LIN {X 0,Y 207.652,Z 346.509,A -85,B 0,C 180,E1 -25427.031,E2 -25427.031} C_VEL
LIN {X 0,Y 210.503,Z 352.306,A -85,B 0,C 180,E1 -25428.836,E2 -25428.836} C_VEL
LIN {X 0,Y 203.288,Z 423.819,A -85,B 0,C 180,E1 -25430.749,E2 -25430.749} C_VEL
LIN {X 0,Y 200.381,Z 440.802,A -85,B 0,C 180,E1 -25431.417,E2 -25431.417} C_VEL
LIN {X 0,Y 196.445,Z 457.536,A -85,B 0,C 180,E1 -25432.38,E2 -25432.38} C_VEL
LIN {X 0,Y 191.604,Z 473.562,A -85,B 0,C 180,E1 -25433.622,E2 -25433.622} C_VEL
LIN {X 0,Y 186.062,Z 488.689,A -85,B 0,C 180,E1 -25435.158,E2 -25435.158} C_VEL
LIN {X 0,Y 179.509,Z 503.688,A -85,B 0,C 180,E1 -25437.096,E2 -25437.096} C_VEL
LIN {X 0,Y 172.547,Z 517.473,A -85,B 0,C 180,E1 -25439.393,E2 -25439.393} C_VEL
LIN {X 0,Y 164.589,Z 531.208,A -85,B 0,C 180,E1 -25442.33,E2 -25442.33} C_VEL
LIN {X 0,Y 157.144,Z 542.82,A -85,B 0,C 180,E1 -25445.563,E2 -25445.563} C_VEL
LIN {X 0,Y 149.721,Z 553.398,A -85,B 0,C 180,E1 -25449.305,E2 -25449.305} C_VEL
LIN {X 0,Y 142.748,Z 562.767,A -85,B 0,C 180,E1 -25453.554,E2 -25453.554} C_VEL
LIN {X 0,Y 136.314,Z 570.972,A -85,B 0,C 180,E1 -25458.403,E2 -25458.403} C_VEL
LIN {X 0,Y 130.699,Z 578.07,A -85,B 0,C 180,E1 -25463.825,E2 -25463.825} C_VEL
LIN {X 0,Y 125.94,Z 584.277,A -85,B 0,C 180,E1 -25469.999,E2 -25469.999} C_VEL
LIN {X 0,Y 122.402,Z 589.195,A -85,B 0,C 180,E1 -25476.593,E2 -25476.593} C_VEL
LIN {X 0,Y 119.976,Z 592.988,A -85,B 0,C 180,E1 -25483.55,E2 -25483.55} C_VEL
LIN {X 0,Y 118.782,Z 595.717,A -85,B 0,C 180,E1 -25490.792,E2 -25490.792} C_VEL
LIN {X 0,Y 118.646,Z 597.115,A -85,B 0,C 180,E1 -25497.312,E2 -25497.312} C_VEL
LIN {X 0,Y 119.339,Z 597.749,A -85,B 0,C 180,E1 -25504.465,E2 -25504.465} C_VEL
LIN {X 0,Y 120.964,Z 597.343,A -85,B 0,C 180,E1 -25510.949,E2 -25510.949} C_VEL
LIN {X 0,Y 123.876,Z 596.092,A -85,B 0,C 180,E1 -25517.521,E2 -25517.521} C_VEL
LIN {X 0,Y 128.898,Z 593.311,A -85,B 0,C 180,E1 -25524.868,E2 -25524.868} C_VEL
LIN {X 0,Y 135.659,Z 589.135,A -85,B 0,C 180,E1 -25531.725,E2 -25531.725} C_VEL
LIN {X 0,Y 144.193,Z 583.478,A -85,B 0,C 180,E1 -25537.826,E2 -25537.826} C_VEL
LIN {X 0,Y 152.82,Z 577.234,A -85,B 0,C 180,E1 -25542.598,E2 -25542.598} C_VEL
LIN {X 0,Y 163.268,Z 568.849,A -85,B 0,C 180,E1 -25547.195,E2 -25547.195} C_VEL
LIN {X 0,Y 174.835,Z 558.387,A -85,B 0,C 180,E1 -25551.263,E2 -25551.263} C_VEL
LIN {X 0,Y 185.382,Z 547.58,A -85,B 0,C 180,E1 -25554.346,E2 -25554.346} C_VEL
LIN {X 0,Y 195.153,Z 536.256,A -85,B 0,C 180,E1 -25556.791,E2 -25556.791} C_VEL
LIN {X 0,Y 204.724,Z 523.645,A -85,B 0,C 180,E1 -25558.892,E2 -25558.892} C_VEL
LIN {X 0,Y 213.483,Z 510.379,A -85,B 0,C 180,E1 -25560.609,E2 -25560.609} C_VEL
LIN {X 0,Y 220.417,Z 498.375,A -85,B 0,C 180,E1 -25561.827,E2 -25561.827} C_VEL
LIN {X 0,Y 227.397,Z 484.222,A -85,B 0,C 180,E1 -25562.988,E2 -25562.988} C_VEL
LIN {X 0,Y 233.808,Z 468.556,A -85,B 0,C 180,E1 -25564.007,E2 -25564.007} C_VEL
LIN {X 0,Y 239.121,Z 452.344,A -85,B 0,C 180,E1 -25564.783,E2 -25564.783} C_VEL
LIN {X 0,Y 243.235,Z 435.804,A -85,B 0,C 180,E1 -25565.349,E2 -25565.349} C_VEL
LIN {X 0,Y 246.105,Z 418.602,A -85,B 0,C 180,E1 -25565.773,E2 -25565.773} C_VEL
LIN {X 0,Y 251.259,Z 376.905,A -85,B 0,C 180,E1 -25566.684,E2 -25566.684} C_VEL
LIN {X 0,Y 250.782,Z 375.19,A -85,B 0,C 180,E1 -25568.055,E2 -25568.055} C_VEL
LIN {X 0,Y 250.079,Z 372.447,A -85,B 0,C 180,E1 -25572.163,E2 -25572.163} C_VEL
LIN {X 0,Y 250.037,Z 372.701,A -85,B 0,C 180,E1 -25573.31,E2 -25573.31} C_VEL
LIN {X 0,Y 250.756,Z 375.692,A -85,B 0,C 180,E1 -25577.654,E2 -25577.654} C_VEL
LIN {X 0,Y 251.253,Z 377.3,A -85,B 0,C 180,E1 -25579.03,E2 -25579.03} C_VEL
LIN {X 0,Y 244.616,Z 429.393,A -85,B 0,C 180,E1 -25580.146,E2 -25580.146} C_VEL
LIN {X 0,Y 241.029,Z 446.475,A -85,B 0,C 180,E1 -25580.592,E2 -25580.592} C_VEL
LIN {X 0,Y 236.395,Z 462.41,A -85,B 0,C 180,E1 -25581.149,E2 -25581.149} C_VEL
LIN {X 0,Y 230.959,Z 477.274,A -85,B 0,C 180,E1 -25581.862,E2 -25581.862} C_VEL
LIN {X 0,Y 224.757,Z 491.347,A -85,B 0,C 180,E1 -25582.717,E2 -25582.717} C_VEL
LIN {X 0,Y 217.928,Z 504.427,A -85,B 0,C 180,E1 -25583.787,E2 -25583.787} C_VEL
LIN {X 0,Y 208.905,Z 519.27,A -85,B 0,C 180,E1 -25585.296,E2 -25585.296} C_VEL
LIN {X 0,Y 200.844,Z 530.92,A -85,B 0,C 180,E1 -25586.838,E2 -25586.838} C_VEL
LIN {X 0,Y 190.88,Z 543.575,A -85,B 0,C 180,E1 -25589.023,E2 -25589.023} C_VEL
LIN {X 0,Y 181.232,Z 554.346,A -85,B 0,C 180,E1 -25591.448,E2 -25591.448} C_VEL
LIN {X 0,Y 170.694,Z 564.923,A -85,B 0,C 180,E1 -25594.57,E2 -25594.57} C_VEL
LIN {X 0,Y 169.098,Z 566.423,A -85,B 0,C 180,E1 -25595.081,E2 -25595.081} C_VEL
LIN {X 0,Y 165.201,Z 569.732,A -85,B 0,C 180,E1 -25596.102,E2 -25596.102} C_VEL
LIN {X 0,Y 157.698,Z 574.973,A -85,B 0,C 180,E1 -25597.464,E2 -25597.464} C_VEL
LIN {X 0,Y 150.146,Z 579.765,A -85,B 0,C 180,E1 -25599.042,E2 -25599.042} C_VEL
LIN {X 0,Y 146.248,Z 582.367,A -85,B 0,C 180,E1 -25600.426,E2 -25600.426} C_VEL
LIN {X 0,Y 136.237,Z 589.443,A -85,B 0,C 180,E1 -25605.862,E2 -25605.862} C_VEL
LIN {X 0,Y 128.84,Z 594.26,A -85,B 0,C 180,E1 -25611.15,E2 -25611.15} C_VEL
LIN {X 0,Y 121.309,Z 598.92,A -85,B 0,C 180,E1 -25618.575,E2 -25618.575} C_VEL
LIN {X 0,Y 116.893,Z 601.559,A -85,B 0,C 180,E1 -25625.112,E2 -25625.112} C_VEL
LIN {X 0,Y 113.834,Z 603.26,A -85,B 0,C 180,E1 -25632.021,E2 -25632.021} C_VEL
LIN {X 0,Y 112.343,Z 604.035,A -85,B 0,C 180,E1 -25639.184,E2 -25639.184} C_VEL
LIN {X 0,Y 112.095,Z 603.898,A -85,B 0,C 180,E1 -25646.406,E2 -25646.406} C_VEL
LIN {X 0,Y 112.259,Z 603.468,A -85,B 0,C 180,E1 -25650.001,E2 -25650.001} C_VEL
LIN {X 0,Y 112.154,Z 602.73,A -85,B 0,C 180,E1 -25653.594,E2 -25653.594} C_VEL
LIN {X 0,Y 112.377,Z 600.537,A -85,B 0,C 180,E1 -25660.815,E2 -25660.815} C_VEL
LIN {X 0,Y 113.815,Z 597.25,A -85,B 0,C 180,E1 -25667.985,E2 -25667.985} C_VEL
LIN {X 0,Y 116.648,Z 592.834,A -85,B 0,C 180,E1 -25674.946,E2 -25674.946} C_VEL
LIN {X 0,Y 120.876,Z 587.27,A -85,B 0,C 180,E1 -25681.553,E2 -25681.553} C_VEL
LIN {X 0,Y 126.437,Z 580.31,A -85,B 0,C 180,E1 -25687.694,E2 -25687.694} C_VEL
LIN {X 0,Y 133.293,Z 571.931,A -85,B 0,C 180,E1 -25693.27,E2 -25693.27} C_VEL
LIN {X 0,Y 141.317,Z 561.914,A -85,B 0,C 180,E1 -25698.244,E2 -25698.244} C_VEL
LIN {X 0,Y 148.682,Z 551.934,A -85,B 0,C 180,E1 -25702.085,E2 -25702.085} C_VEL
LIN {X 0,Y 157.311,Z 539.305,A -85,B 0,C 180,E1 -25705.741,E2 -25705.741} C_VEL
LIN {X 0,Y 165.607,Z 525.855,A -85,B 0,C 180,E1 -25708.656,E2 -25708.656} C_VEL
LIN {X 0,Y 172.473,Z 513.183,A -85,B 0,C 180,E1 -25710.8,E2 -25710.8} C_VEL
LIN {X 0,Y 179.768,Z 497.842,A -85,B 0,C 180,E1 -25712.799,E2 -25712.799} C_VEL
LIN {X 0,Y 185.354,Z 483.986,A -85,B 0,C 180,E1 -25714.226,E2 -25714.226} C_VEL
LIN {X 0,Y 190.733,Z 468.038,A -85,B 0,C 180,E1 -25715.46,E2 -25715.46} C_VEL
LIN {X 0,Y 194.945,Z 452.39,A -85,B 0,C 180,E1 -25716.337,E2 -25716.337} C_VEL
LIN {X 0,Y 198.282,Z 436,A -85,B 0,C 180,E1 -25716.992,E2 -25716.992} C_VEL
LIN {X 0,Y 200.576,Z 417.694,A -85,B 0,C 180,E1 -25717.565,E2 -25717.565} C_VEL
LIN {X 0,Y 206.676,Z 357.209,A -85,B 0,C 180,E1 -25719.155,E2 -25719.155} C_VEL
LIN {X 0,Y 203.434,Z 349.128,A -85,B 0,C 180,E1 -25721.494,E2 -25721.494} C_VEL
LIN {X 0,Y 198.655,Z 340.024,A -85,B 0,C 180,E1 -25725.138,E2 -25725.138} C_VEL
LIN {X 0,Y 195.269,Z 333.943,A -85,B 0,C 180,E1 -25728.08,E2 -25728.08} C_VEL
LIN {X 0,Y 192.367,Z 328.903,A -85,B 0,C 180,E1 -25730.999,E2 -25730.999} C_VEL
LIN {X 0,Y 189.117,Z 323.394,A -85,B 0,C 180,E1 -25734.828,E2 -25734.828} C_VEL
LIN {X 0,Y 186.858,Z 319.626,A -85,B 0,C 180,E1 -25738.137,E2 -25738.137} C_VEL
LIN {X 0,Y 184.729,Z 315.82,A -85,B 0,C 180,E1 -25742.307,E2 -25742.307} C_VEL
LIN {X 0,Y 184.223,Z 315.108,A -85,B 0,C 180,E1 -25743.467,E2 -25743.467} C_VEL
LIN {X 0,Y 182.713,Z 313.172,A -85,B 0,C 180,E1 -25748.571,E2 -25748.571} C_VEL
LIN {X 0,Y 182.415,Z 311.657,A -85,B 0,C 180,E1 -25752.151,E2 -25752.151} C_VEL
LIN {X 0,Y 182.382,Z 311.95,A -85,B 0,C 180,E1 -25754.436,E2 -25754.436} C_VEL
LIN {X 0,Y 183.988,Z 315.501,A -85,B 0,C 180,E1 -25762.686,E2 -25762.686} C_VEL
LIN {X 0,Y 184.724,Z 316.384,A -85,B 0,C 180,E1 -25764.365,E2 -25764.365} C_VEL
LIN {X 0,Y 187.441,Z 320.995,A -85,B 0,C 180,E1 -25769.378,E2 -25769.378} C_VEL
LIN {X 0,Y 190.002,Z 325.194,A -85,B 0,C 180,E1 -25772.883,E2 -25772.883} C_VEL
LIN {X 0,Y 193.097,Z 330.301,A -85,B 0,C 180,E1 -25776.321,E2 -25776.321} C_VEL
LIN {X 0,Y 197.341,Z 337.624,A -85,B 0,C 180,E1 -25780.284,E2 -25780.284} C_VEL
LIN {X 0,Y 202.688,Z 347.63,A -85,B 0,C 180,E1 -25784.496,E2 -25784.496} C_VEL
LIN {X 0,Y 206.664,Z 355.706,A -85,B 0,C 180,E1 -25787.241,E2 -25787.241} C_VEL
LIN {X 0,Y 199.416,Z 424.921,A -85,B 0,C 180,E1 -25789.058,E2 -25789.058} C_VEL
LIN {X 0,Y 196.238,Z 442.746,A -85,B 0,C 180,E1 -25789.777,E2 -25789.777} C_VEL
LIN {X 0,Y 192.185,Z 459.017,A -85,B 0,C 180,E1 -25790.721,E2 -25790.721} C_VEL
LIN {X 0,Y 187.194,Z 474.829,A -85,B 0,C 180,E1 -25791.956,E2 -25791.956} C_VEL
LIN {X 0,Y 181.535,Z 489.677,A -85,B 0,C 180,E1 -25793.471,E2 -25793.471} C_VEL
LIN {X 0,Y 174.797,Z 504.536,A -85,B 0,C 180,E1 -25795.395,E2 -25795.395} C_VEL
LIN {X 0,Y 167.766,Z 518.005,A -85,B 0,C 180,E1 -25797.639,E2 -25797.639} C_VEL
LIN {X 0,Y 160.036,Z 530.9,A -85,B 0,C 180,E1 -25800.393,E2 -25800.393} C_VEL
LIN {X 0,Y 152.843,Z 541.768,A -85,B 0,C 180,E1 -25803.363,E2 -25803.363} C_VEL
LIN {X 0,Y 144.749,Z 552.984,A -85,B 0,C 180,E1 -25807.295,E2 -25807.295} C_VEL
LIN {X 0,Y 136.71,Z 563.26,A -85,B 0,C 180,E1 -25812.034,E2 -25812.034} C_VEL
LIN {X 0,Y 129.48,Z 572.063,A -85,B 0,C 180,E1 -25817.46,E2 -25817.46} C_VEL
LIN {X 0,Y 123.401,Z 579.326,A -85,B 0,C 180,E1 -25823.459,E2 -25823.459} C_VEL
LIN {X 0,Y 118.554,Z 585.3,A -85,B 0,C 180,E1 -25829.999,E2 -25829.999} C_VEL
LIN {X 0,Y 114.968,Z 590.109,A -85,B 0,C 180,E1 -25837.021,E2 -25837.021} C_VEL
LIN {X 0,Y 112.606,Z 593.693,A -85,B 0,C 180,E1 -25844.456,E2 -25844.456} C_VEL
LIN {X 0,Y 111.836,Z 595.471,A -85,B 0,C 180,E1 -25849.502,E2 -25849.502} C_VEL
LIN {X 0,Y 111.555,Z 597.357,A -85,B 0,C 180,E1 -25858.115,E2 -25858.115} C_VEL
LIN {X 0,Y 112.415,Z 597.959,A -85,B 0,C 180,E1 -25865.636,E2 -25865.636} C_VEL
LIN {X 0,Y 114.335,Z 597.539,A -85,B 0,C 180,E1 -25872.542,E2 -25872.542} C_VEL
LIN {X 0,Y 118.302,Z 595.932,A -85,B 0,C 180,E1 -25880.558,E2 -25880.558} C_VEL
LIN {X 0,Y 124.144,Z 593.005,A -85,B 0,C 180,E1 -25888.119,E2 -25888.119} C_VEL
LIN {X 0,Y 131.806,Z 588.593,A -85,B 0,C 180,E1 -25895.016,E2 -25895.016} C_VEL
LIN {X 0,Y 141.166,Z 582.701,A -85,B 0,C 180,E1 -25901.066,E2 -25901.066} C_VEL
LIN {X 0,Y 151.88,Z 575.162,A -85,B 0,C 180,E1 -25906.34,E2 -25906.34} C_VEL
LIN {X 0,Y 162.15,Z 567.093,A -85,B 0,C 180,E1 -25910.309,E2 -25910.309} C_VEL
LIN {X 0,Y 173.171,Z 557.354,A -85,B 0,C 180,E1 -25913.873,E2 -25913.873} C_VEL
LIN {X 0,Y 183.061,Z 547.566,A -85,B 0,C 180,E1 -25916.523,E2 -25916.523} C_VEL
LIN {X 0,Y 193.3,Z 535.996,A -85,B 0,C 180,E1 -25918.912,E2 -25918.912} C_VEL
LIN {X 0,Y 203.056,Z 523.461,A -85,B 0,C 180,E1 -25920.91,E2 -25920.91} C_VEL
LIN {X 0,Y 211.921,Z 510.362,A -85,B 0,C 180,E1 -25922.536,E2 -25922.536} C_VEL
LIN {X 0,Y 219.769,Z 496.993,A -85,B 0,C 180,E1 -25923.801,E2 -25923.801} C_VEL
LIN {X 0,Y 227.299,Z 481.61,A -85,B 0,C 180,E1 -25924.97,E2 -25924.97} C_VEL
LIN {X 0,Y 233.568,Z 466.034,A -85,B 0,C 180,E1 -25925.864,E2 -25925.864} C_VEL
LIN {X 0,Y 238.605,Z 450.348,A -85,B 0,C 180,E1 -25926.553,E2 -25926.553} C_VEL
LIN {X 0,Y 242.42,Z 434.847,A -85,B 0,C 180,E1 -25927.037,E2 -25927.037} C_VEL
LIN {X 0,Y 245.308,Z 417.581,A -85,B 0,C 180,E1 -25927.434,E2 -25927.434} C_VEL
LIN {X 0,Y 249.773,Z 382.182,A -85,B 0,C 180,E1 -25928.18,E2 -25928.18} C_VEL
LIN {X 0,Y 249.115,Z 379.534,A -85,B 0,C 180,E1 -25932.211,E2 -25932.211} C_VEL
LIN {X 0,Y 249.072,Z 380.047,A -85,B 0,C 180,E1 -25933.68,E2 -25933.68} C_VEL
LIN {X 0,Y 249.662,Z 382.544,A -85,B 0,C 180,E1 -25937.298,E2 -25937.298} C_VEL
LIN {X 0,Y 249.721,Z 382.826,A -85,B 0,C 180,E1 -25937.517,E2 -25937.517} C_VEL
LIN {X 0,Y 243.632,Z 429.235,A -85,B 0,C 180,E1 -25938.491,E2 -25938.491} C_VEL
LIN {X 0,Y 239.964,Z 446.328,A -85,B 0,C 180,E1 -25938.916,E2 -25938.916} C_VEL
LIN {X 0,Y 235.154,Z 462.482,A -85,B 0,C 180,E1 -25939.445,E2 -25939.445} C_VEL
LIN {X 0,Y 229.275,Z 478.077,A -85,B 0,C 180,E1 -25940.16,E2 -25940.16} C_VEL
LIN {X 0,Y 222.96,Z 491.964,A -85,B 0,C 180,E1 -25940.965,E2 -25940.965} C_VEL
LIN {X 0,Y 215.992,Z 504.967,A -85,B 0,C 180,E1 -25941.98,E2 -25941.98} C_VEL
LIN {X 0,Y 207.556,Z 518.518,A -85,B 0,C 180,E1 -25943.3,E2 -25943.3} C_VEL
LIN {X 0,Y 197.782,Z 532.101,A -85,B 0,C 180,E1 -25945.029,E2 -25945.029} C_VEL
LIN {X 0,Y 187.573,Z 544.548,A -85,B 0,C 180,E1 -25947.146,E2 -25947.146} C_VEL
LIN {X 0,Y 177.657,Z 555.179,A -85,B 0,C 180,E1 -25949.509,E2 -25949.509} C_VEL
LIN {X 0,Y 166.777,Z 565.552,A -85,B 0,C 180,E1 -25952.565,E2 -25952.565} C_VEL
LIN {X 0,Y 156.514,Z 574.365,A -85,B 0,C 180,E1 -25956.076,E2 -25956.076} C_VEL
LIN {X 0,Y 146.248,Z 582.367,A -85,B 0,C 180,E1 -25960.426,E2 -25960.426} C_VEL
LIN {X 0,Y 142.37,Z 584.882,A -85,B 0,C 180,E1 -25961.909,E2 -25961.909} C_VEL
LIN {X 0,Y 128.864,Z 591.543,A -85,B 0,C 180,E1 -25965.963,E2 -25965.963} C_VEL
LIN {X 0,Y 125.038,Z 593.438,A -85,B 0,C 180,E1 -25967.8,E2 -25967.8} C_VEL
LIN {X 0,Y 124,Z 593.996,A -85,B 0,C 180,E1 -25968.519,E2 -25968.519} C_VEL
LIN {X 0,Y 118.221,Z 597.304,A -85,B 0,C 180,E1 -25973.526,E2 -25973.526} C_VEL
LIN {X 0,Y 111.139,Z 601.108,A -85,B 0,C 180,E1 -25982.288,E2 -25982.288} C_VEL
LIN {X 0,Y 107.047,Z 603.123,A -85,B 0,C 180,E1 -25990.838,E2 -25990.838} C_VEL
LIN {X 0,Y 105.316,Z 603.849,A -85,B 0,C 180,E1 -25998.453,E2 -25998.453} C_VEL
LIN {X 0,Y 105.003,Z 603.625,A -85,B 0,C 180,E1 -26006.163,E2 -26006.163} C_VEL
LIN {X 0,Y 105.171,Z 603.188,A -85,B 0,C 180,E1 -26010.001,E2 -26010.001} C_VEL
LIN {X 0,Y 105.044,Z 602.411,A -85,B 0,C 180,E1 -26013.837,E2 -26013.837} C_VEL
LIN {X 0,Y 105.342,Z 600.124,A -85,B 0,C 180,E1 -26021.547,E2 -26021.547} C_VEL
LIN {X 0,Y 107.025,Z 596.791,A -85,B 0,C 180,E1 -26029.169,E2 -26029.169} C_VEL
LIN {X 0,Y 110.361,Z 591.985,A -85,B 0,C 180,E1 -26036.932,E2 -26036.932} C_VEL
LIN {X 0,Y 114.752,Z 586.607,A -85,B 0,C 180,E1 -26043.45,E2 -26043.45} C_VEL
LIN {X 0,Y 120.785,Z 579.582,A -85,B 0,C 180,E1 -26049.796,E2 -26049.796} C_VEL
LIN {X 0,Y 128.11,Z 571.079,A -85,B 0,C 180,E1 -26055.494,E2 -26055.494} C_VEL
LIN {X 0,Y 135.485,Z 562.316,A -85,B 0,C 180,E1 -26059.918,E2 -26059.918} C_VEL
LIN {X 0,Y 143.59,Z 551.812,A -85,B 0,C 180,E1 -26064.032,E2 -26064.032} C_VEL
LIN {X 0,Y 152.073,Z 539.897,A -85,B 0,C 180,E1 -26067.503,E2 -26067.503} C_VEL
LIN {X 0,Y 159.946,Z 527.695,A -85,B 0,C 180,E1 -26070.205,E2 -26070.205} C_VEL
LIN {X 0,Y 167.959,Z 513.568,A -85,B 0,C 180,E1 -26072.638,E2 -26072.638} C_VEL
LIN {X 0,Y 175.147,Z 499.029,A -85,B 0,C 180,E1 -26074.534,E2 -26074.534} C_VEL
LIN {X 0,Y 181.6,Z 483.516,A -85,B 0,C 180,E1 -26076.106,E2 -26076.106} C_VEL
LIN {X 0,Y 187.103,Z 467.528,A -85,B 0,C 180,E1 -26077.312,E2 -26077.312} C_VEL
LIN {X 0,Y 191.271,Z 452.324,A -85,B 0,C 180,E1 -26078.14,E2 -26078.14} C_VEL
LIN {X 0,Y 194.844,Z 435.104,A -85,B 0,C 180,E1 -26078.796,E2 -26078.796} C_VEL
LIN {X 0,Y 197.455,Z 413.787,A -85,B 0,C 180,E1 -26079.439,E2 -26079.439} C_VEL
LIN {X 0,Y 203.035,Z 360.3,A -85,B 0,C 180,E1 -26080.802,E2 -26080.802} C_VEL
LIN {X 0,Y 200.193,Z 353.501,A -85,B 0,C 180,E1 -26082.948,E2 -26082.948} C_VEL
LIN {X 0,Y 195.688,Z 344.623,A -85,B 0,C 180,E1 -26086.67,E2 -26086.67} C_VEL
LIN {X 0,Y 191.781,Z 337.326,A -85,B 0,C 180,E1 -26090.466,E2 -26090.466} C_VEL
LIN {X 0,Y 188.334,Z 331.299,A -85,B 0,C 180,E1 -26094.477,E2 -26094.477} C_VEL
LIN {X 0,Y 185.551,Z 326.428,A -85,B 0,C 180,E1 -26098.624,E2 -26098.624} C_VEL
LIN {X 0,Y 183.466,Z 322.485,A -85,B 0,C 180,E1 -26102.96,E2 -26102.96} C_VEL
LIN {X 0,Y 181.576,Z 319.623,A -85,B 0,C 180,E1 -26109.861,E2 -26109.861} C_VEL
LIN {X 0,Y 181.462,Z 318.692,A -85,B 0,C 180,E1 -26112.216,E2 -26112.216} C_VEL
LIN {X 0,Y 181.428,Z 318.945,A -85,B 0,C 180,E1 -26114.194,E2 -26114.194} C_VEL
LIN {X 0,Y 182.981,Z 322.533,A -85,B 0,C 180,E1 -26122.587,E2 -26122.587} C_VEL
LIN {X 0,Y 183.549,Z 323.299,A -85,B 0,C 180,E1 -26123.951,E2 -26123.951} C_VEL
LIN {X 0,Y 185.98,Z 327.563,A -85,B 0,C 180,E1 -26128.691,E2 -26128.691} C_VEL
LIN {X 0,Y 188.437,Z 331.784,A -85,B 0,C 180,E1 -26132.228,E2 -26132.228} C_VEL
LIN {X 0,Y 191.744,Z 337.443,A -85,B 0,C 180,E1 -26136.04,E2 -26136.04} C_VEL
LIN {X 0,Y 195.587,Z 344.406,A -85,B 0,C 180,E1 -26139.765,E2 -26139.765} C_VEL
LIN {X 0,Y 200.518,Z 354.128,A -85,B 0,C 180,E1 -26143.815,E2 -26143.815} C_VEL
LIN {X 0,Y 202.955,Z 359.352,A -85,B 0,C 180,E1 -26145.606,E2 -26145.606} C_VEL
LIN {X 0,Y 195.85,Z 425.055,A -85,B 0,C 180,E1 -26147.278,E2 -26147.278} C_VEL
LIN {X 0,Y 192.598,Z 442.897,A -85,B 0,C 180,E1 -26147.981,E2 -26147.981} C_VEL
LIN {X 0,Y 188.451,Z 459.179,A -85,B 0,C 180,E1 -26148.906,E2 -26148.906} C_VEL
LIN {X 0,Y 183.495,Z 474.57,A -85,B 0,C 180,E1 -26150.082,E2 -26150.082} C_VEL
LIN {X 0,Y 177.172,Z 490.667,A -85,B 0,C 180,E1 -26151.698,E2 -26151.698} C_VEL
LIN {X 0,Y 170.239,Z 505.391,A -85,B 0,C 180,E1 -26153.598,E2 -26153.598} C_VEL
LIN {X 0,Y 162.857,Z 519.006,A -85,B 0,C 180,E1 -26155.874,E2 -26155.874} C_VEL
LIN {X 0,Y 155.024,Z 531.598,A -85,B 0,C 180,E1 -26158.577,E2 -26158.577} C_VEL
LIN {X 0,Y 147.573,Z 542.388,A -85,B 0,C 180,E1 -26161.56,E2 -26161.56} C_VEL
LIN {X 0,Y 139.389,Z 553.267,A -85,B 0,C 180,E1 -26165.429,E2 -26165.429} C_VEL
LIN {X 0,Y 131.819,Z 562.557,A -85,B 0,C 180,E1 -26169.723,E2 -26169.723} C_VEL
LIN {X 0,Y 124.501,Z 571.025,A -85,B 0,C 180,E1 -26174.922,E2 -26174.922} C_VEL
LIN {X 0,Y 117.552,Z 578.899,A -85,B 0,C 180,E1 -26181.403,E2 -26181.403} C_VEL
LIN {X 0,Y 112.529,Z 584.729,A -85,B 0,C 180,E1 -26187.818,E2 -26187.818} C_VEL
LIN {X 0,Y 108.333,Z 589.896,A -85,B 0,C 180,E1 -26195.583,E2 -26195.583} C_VEL
LIN {X 0,Y 106.221,Z 592.816,A -85,B 0,C 180,E1 -26201.448,E2 -26201.448} C_VEL
LIN {X 0,Y 104.685,Z 595.791,A -85,B 0,C 180,E1 -26209.968,E2 -26209.968} C_VEL
LIN {X 0,Y 104.484,Z 597.598,A -85,B 0,C 180,E1 -26219.022,E2 -26219.022} C_VEL
LIN {X 0,Y 105.543,Z 598.171,A -85,B 0,C 180,E1 -26226.959,E2 -26226.959} C_VEL
LIN {X 0,Y 108.301,Z 597.606,A -85,B 0,C 180,E1 -26235.545,E2 -26235.545} C_VEL
LIN {X 0,Y 113.083,Z 595.764,A -85,B 0,C 180,E1 -26243.892,E2 -26243.892} C_VEL
LIN {X 0,Y 120.403,Z 592.298,A -85,B 0,C 180,E1 -26252.163,E2 -26252.163} C_VEL
LIN {X 0,Y 128.424,Z 588.03,A -85,B 0,C 180,E1 -26258.481,E2 -26258.481} C_VEL
LIN {X 0,Y 138.623,Z 581.936,A -85,B 0,C 180,E1 -26264.418,E2 -26264.418} C_VEL
LIN {X 0,Y 150.095,Z 574.166,A -85,B 0,C 180,E1 -26269.505,E2 -26269.505} C_VEL
LIN {X 0,Y 161.272,Z 565.57,A -85,B 0,C 180,E1 -26273.416,E2 -26273.416} C_VEL
LIN {X 0,Y 172.475,Z 555.804,A -85,B 0,C 180,E1 -26276.659,E2 -26276.659} C_VEL
LIN {X 0,Y 183.978,Z 544.43,A -85,B 0,C 180,E1 -26279.434,E2 -26279.434} C_VEL
LIN {X 0,Y 194.577,Z 532.419,A -85,B 0,C 180,E1 -26281.631,E2 -26281.631} C_VEL
LIN {X 0,Y 204.162,Z 519.965,A -85,B 0,C 180,E1 -26283.38,E2 -26283.38} C_VEL
LIN {X 0,Y 213.276,Z 506.154,A -85,B 0,C 180,E1 -26284.878,E2 -26284.878} C_VEL
LIN {X 0,Y 221.766,Z 491.023,A -85,B 0,C 180,E1 -26286.128,E2 -26286.128} C_VEL
LIN {X 0,Y 228.552,Z 476.498,A -85,B 0,C 180,E1 -26287.065,E2 -26287.065} C_VEL
LIN {X 0,Y 234.435,Z 461.157,A -85,B 0,C 180,E1 -26287.837,E2 -26287.837} C_VEL
LIN {X 0,Y 239.215,Z 445.35,A -85,B 0,C 180,E1 -26288.429,E2 -26288.429} C_VEL
LIN {X 0,Y 242.999,Z 428.02,A -85,B 0,C 180,E1 -26288.867,E2 -26288.867} C_VEL
LIN {X 0,Y 248.346,Z 388.428,A -85,B 0,C 180,E1 -26289.704,E2 -26289.704} C_VEL
LIN {X 0,Y 248.154,Z 386.601,A -85,B 0,C 180,E1 -26292.259,E2 -26292.259} C_VEL
LIN {X 0,Y 248.107,Z 387.202,A -85,B 0,C 180,E1 -26293.734,E2 -26293.734} C_VEL
LIN {X 0,Y 248.335,Z 388.591,A -85,B 0,C 180,E1 -26295.976,E2 -26295.976} C_VEL
LIN {X 0,Y 242.921,Z 428.909,A -85,B 0,C 180,E1 -26296.817,E2 -26296.817} C_VEL
LIN {X 0,Y 239.104,Z 446.428,A -85,B 0,C 180,E1 -26297.228,E2 -26297.228} C_VEL
LIN {X 0,Y 233.844,Z 463.654,A -85,B 0,C 180,E1 -26297.764,E2 -26297.764} C_VEL
LIN {X 0,Y 227.801,Z 479.082,A -85,B 0,C 180,E1 -26298.439,E2 -26298.439} C_VEL
LIN {X 0,Y 220.58,Z 494.192,A -85,B 0,C 180,E1 -26299.287,E2 -26299.287} C_VEL
LIN {X 0,Y 212.729,Z 508.137,A -85,B 0,C 180,E1 -26300.379,E2 -26300.379} C_VEL
LIN {X 0,Y 203.365,Z 522.314,A -85,B 0,C 180,E1 -26301.761,E2 -26301.761} C_VEL
LIN {X 0,Y 194.928,Z 533.357,A -85,B 0,C 180,E1 -26303.167,E2 -26303.167} C_VEL
LIN {X 0,Y 184.475,Z 545.538,A -85,B 0,C 180,E1 -26305.205,E2 -26305.205} C_VEL
LIN {X 0,Y 175.719,Z 554.579,A -85,B 0,C 180,E1 -26307.142,E2 -26307.142} C_VEL
LIN {X 0,Y 165.846,Z 563.8,A -85,B 0,C 180,E1 -26309.693,E2 -26309.693} C_VEL
LIN {X 0,Y 155.33,Z 572.634,A -85,B 0,C 180,E1 -26312.884,E2 -26312.884} C_VEL
LIN {X 0,Y 144.886,Z 580.464,A -85,B 0,C 180,E1 -26316.837,E2 -26316.837} C_VEL
LIN {X 0,Y 135.523,Z 586.874,A -85,B 0,C 180,E1 -26321.243,E2 -26321.243} C_VEL
LIN {X 0,Y 127.701,Z 591.787,A -85,B 0,C 180,E1 -26325.863,E2 -26325.863} C_VEL
LIN {X 0,Y 124,Z 593.996,A -85,B 0,C 180,E1 -26328.519,E2 -26328.519} C_VEL
LIN {X 0,Y 120.636,Z 595.716,A -85,B 0,C 180,E1 -26330.659,E2 -26330.659} C_VEL
LIN {X 0,Y 113.885,Z 598.167,A -85,B 0,C 180,E1 -26334.001,E2 -26334.001} C_VEL
LIN {X 0,Y 108.621,Z 599.802,A -85,B 0,C 180,E1 -26336.951,E2 -26336.951} C_VEL
LIN {X 0,Y 105.515,Z 600.791,A -85,B 0,C 180,E1 -26339.586,E2 -26339.586} C_VEL
LIN {X 0,Y 104.763,Z 601.106,A -85,B 0,C 180,E1 -26340.562,E2 -26340.562} C_VEL
LIN {X 0,Y 100.287,Z 602.987,A -85,B 0,C 180,E1 -26349.49,E2 -26349.49} C_VEL
LIN {X 0,Y 98.32,Z 603.666,A -85,B 0,C 180,E1 -26357.619,E2 -26357.619} C_VEL
LIN {X 0,Y 97.904,Z 603.347,A -85,B 0,C 180,E1 -26365.885,E2 -26365.885} C_VEL
LIN {X 0,Y 98.074,Z 602.871,A -85,B 0,C 180,E1 -26370.001,E2 -26370.001} C_VEL
LIN {X 0,Y 97.935,Z 602.09,A -85,B 0,C 180,E1 -26374.116,E2 -26374.116} C_VEL
LIN {X 0,Y 98.339,Z 599.709,A -85,B 0,C 180,E1 -26382.381,E2 -26382.381} C_VEL
LIN {X 0,Y 100.26,Z 596.325,A -85,B 0,C 180,E1 -26390.518,E2 -26390.518} C_VEL
LIN {X 0,Y 103.733,Z 591.704,A -85,B 0,C 180,E1 -26398.312,E2 -26398.312} C_VEL
LIN {X 0,Y 108.793,Z 585.927,A -85,B 0,C 180,E1 -26405.55,E2 -26405.55} C_VEL
LIN {X 0,Y 115.314,Z 578.84,A -85,B 0,C 180,E1 -26412.099,E2 -26412.099} C_VEL
LIN {X 0,Y 123.149,Z 570.208,A -85,B 0,C 180,E1 -26417.894,E2 -26417.894} C_VEL
LIN {X 0,Y 130.904,Z 561.288,A -85,B 0,C 180,E1 -26422.364,E2 -26422.364} C_VEL
LIN {X 0,Y 138.749,Z 551.57,A -85,B 0,C 180,E1 -26426.139,E2 -26426.139} C_VEL
LIN {X 0,Y 148.288,Z 538.592,A -85,B 0,C 180,E1 -26429.877,E2 -26429.877} C_VEL
LIN {X 0,Y 157.155,Z 525.08,A -85,B 0,C 180,E1 -26432.725,E2 -26432.725} C_VEL
LIN {X 0,Y 164.915,Z 511.515,A -85,B 0,C 180,E1 -26434.903,E2 -26434.903} C_VEL
LIN {X 0,Y 172.15,Z 496.868,A -85,B 0,C 180,E1 -26436.716,E2 -26436.716} C_VEL
LIN {X 0,Y 178.799,Z 480.875,A -85,B 0,C 180,E1 -26438.221,E2 -26438.221} C_VEL
LIN {X 0,Y 184.059,Z 465.508,A -85,B 0,C 180,E1 -26439.308,E2 -26439.308} C_VEL
LIN {X 0,Y 188.467,Z 449.393,A -85,B 0,C 180,E1 -26440.123,E2 -26440.123} C_VEL
LIN {X 0,Y 191.901,Z 431.925,A -85,B 0,C 180,E1 -26440.741,E2 -26440.741} C_VEL
LIN {X 0,Y 195.837,Z 397.362,A -85,B 0,C 180,E1 -26441.659,E2 -26441.659} C_VEL
LIN {X 0,Y 199.417,Z 363.344,A -85,B 0,C 180,E1 -26442.541,E2 -26442.541} C_VEL
LIN {X 0,Y 197.049,Z 357.777,A -85,B 0,C 180,E1 -26444.485,E2 -26444.485} C_VEL
LIN {X 0,Y 192.648,Z 348.842,A -85,B 0,C 180,E1 -26448.427,E2 -26448.427} C_VEL
LIN {X 0,Y 188.938,Z 341.884,A -85,B 0,C 180,E1 -26452.395,E2 -26452.395} C_VEL
LIN {X 0,Y 186.095,Z 336.597,A -85,B 0,C 180,E1 -26456.169,E2 -26456.169} C_VEL
LIN {X 0,Y 184.084,Z 332.968,A -85,B 0,C 180,E1 -26459.427,E2 -26459.427} C_VEL
LIN {X 0,Y 182.164,Z 329.136,A -85,B 0,C 180,E1 -26463.76,E2 -26463.76} C_VEL
LIN {X 0,Y 180.671,Z 326.991,A -85,B 0,C 180,E1 -26469.336,E2 -26469.336} C_VEL
LIN {X 0,Y 180.507,Z 325.726,A -85,B 0,C 180,E1 -26472.282,E2 -26472.282} C_VEL
LIN {X 0,Y 180.464,Z 326.075,A -85,B 0,C 180,E1 -26474.259,E2 -26474.259} C_VEL
LIN {X 0,Y 181.925,Z 329.518,A -85,B 0,C 180,E1 -26482.36,E2 -26482.36} C_VEL
LIN {X 0,Y 182.346,Z 330.102,A -85,B 0,C 180,E1 -26483.428,E2 -26483.428} C_VEL
LIN {X 0,Y 184.753,Z 334.571,A -85,B 0,C 180,E1 -26488.357,E2 -26488.357} C_VEL
LIN {X 0,Y 186.972,Z 338.512,A -85,B 0,C 180,E1 -26491.669,E2 -26491.669} C_VEL
LIN {X 0,Y 190.197,Z 344.272,A -85,B 0,C 180,E1 -26495.556,E2 -26495.556} C_VEL
LIN {X 0,Y 194.09,Z 351.75,A -85,B 0,C 180,E1 -26499.467,E2 -26499.467} C_VEL
LIN {X 0,Y 198.93,Z 361.681,A -85,B 0,C 180,E1 -26503.546,E2 -26503.546} C_VEL
LIN {X 0,Y 199.311,Z 362.515,A -85,B 0,C 180,E1 -26503.842,E2 -26503.842} C_VEL
LIN {X 0,Y 192.572,Z 424.141,A -85,B 0,C 180,E1 -26505.425,E2 -26505.425} C_VEL
LIN {X 0,Y 189.518,Z 440.955,A -85,B 0,C 180,E1 -26506.04,E2 -26506.04} C_VEL
LIN {X 0,Y 185.265,Z 457.835,A -85,B 0,C 180,E1 -26506.935,E2 -26506.935} C_VEL
LIN {X 0,Y 180.162,Z 473.635,A -85,B 0,C 180,E1 -26508.084,E2 -26508.084} C_VEL
LIN {X 0,Y 174.38,Z 488.378,A -85,B 0,C 180,E1 -26509.487,E2 -26509.487} C_VEL
LIN {X 0,Y 167.269,Z 503.482,A -85,B 0,C 180,E1 -26511.318,E2 -26511.318} C_VEL
LIN {X 0,Y 159.62,Z 517.36,A -85,B 0,C 180,E1 -26513.53,E2 -26513.53} C_VEL
LIN {X 0,Y 151.516,Z 530.207,A -85,B 0,C 180,E1 -26516.178,E2 -26516.178} C_VEL
LIN {X 0,Y 143.718,Z 541.273,A -85,B 0,C 180,E1 -26519.105,E2 -26519.105} C_VEL
LIN {X 0,Y 135.472,Z 551.968,A -85,B 0,C 180,E1 -26522.776,E2 -26522.776} C_VEL
LIN {X 0,Y 127.165,Z 561.76,A -85,B 0,C 180,E1 -26527.24,E2 -26527.24} C_VEL
LIN {X 0,Y 118.919,Z 570.87,A -85,B 0,C 180,E1 -26532.812,E2 -26532.812} C_VEL
LIN {X 0,Y 111.85,Z 578.453,A -85,B 0,C 180,E1 -26539.134,E2 -26539.134} C_VEL
LIN {X 0,Y 106.109,Z 584.712,A -85,B 0,C 180,E1 -26546.201,E2 -26546.201} C_VEL
LIN {X 0,Y 101.732,Z 589.665,A -85,B 0,C 180,E1 -26553.96,E2 -26553.96} C_VEL
LIN {X 0,Y 98.81,Z 593.507,A -85,B 0,C 180,E1 -26562.319,E2 -26562.319} C_VEL
LIN {X 0,Y 97.452,Z 596.275,A -85,B 0,C 180,E1 -26571.135,E2 -26571.135} C_VEL
LIN {X 0,Y 97.451,Z 597.866,A -85,B 0,C 180,E1 -26580.318,E2 -26580.318} C_VEL
LIN {X 0,Y 99.019,Z 598.353,A -85,B 0,C 180,E1 -26589.699,E2 -26589.699} C_VEL
LIN {X 0,Y 102.592,Z 597.649,A -85,B 0,C 180,E1 -26598.896,E2 -26598.896} C_VEL
LIN {X 0,Y 108.268,Z 595.607,A -85,B 0,C 180,E1 -26607.548,E2 -26607.548} C_VEL
LIN {X 0,Y 115.985,Z 592.212,A -85,B 0,C 180,E1 -26615.351,E2 -26615.351} C_VEL
LIN {X 0,Y 125.531,Z 587.402,A -85,B 0,C 180,E1 -26622.126,E2 -26622.126} C_VEL
LIN {X 0,Y 133.694,Z 582.835,A -85,B 0,C 180,E1 -26626.527,E2 -26626.527} C_VEL
LIN {X 0,Y 144.217,Z 576.202,A -85,B 0,C 180,E1 -26631.059,E2 -26631.059} C_VEL
LIN {X 0,Y 155.242,Z 568.397,A -85,B 0,C 180,E1 -26634.834,E2 -26634.834} C_VEL
LIN {X 0,Y 166.297,Z 559.55,A -85,B 0,C 180,E1 -26637.999,E2 -26637.999} C_VEL
LIN {X 0,Y 177.464,Z 549.345,A -85,B 0,C 180,E1 -26640.65,E2 -26640.65} C_VEL
LIN {X 0,Y 188.512,Z 537.807,A -85,B 0,C 180,E1 -26642.908,E2 -26642.908} C_VEL
LIN {X 0,Y 199.233,Z 524.952,A -85,B 0,C 180,E1 -26644.794,E2 -26644.794} C_VEL
LIN {X 0,Y 208.647,Z 511.886,A -85,B 0,C 180,E1 -26646.287,E2 -26646.287} C_VEL
LIN {X 0,Y 216.971,Z 498.411,A -85,B 0,C 180,E1 -26647.444,E2 -26647.444} C_VEL
LIN {X 0,Y 224.701,Z 483.496,A -85,B 0,C 180,E1 -26648.462,E2 -26648.462} C_VEL
LIN {X 0,Y 231.058,Z 468.687,A -85,B 0,C 180,E1 -26649.25,E2 -26649.25} C_VEL
LIN {X 0,Y 236.467,Z 453.114,A -85,B 0,C 180,E1 -26649.884,E2 -26649.884} C_VEL
LIN {X 0,Y 240.629,Z 437.476,A -85,B 0,C 180,E1 -26650.33,E2 -26650.33} C_VEL
LIN {X 0,Y 243.802,Z 420.005,A -85,B 0,C 180,E1 -26650.7,E2 -26650.7} C_VEL
LIN {X 0,Y 247.195,Z 394.564,A -85,B 0,C 180,E1 -26651.207,E2 -26651.207} C_VEL
LIN {X 0,Y 247.181,Z 393.752,A -85,B 0,C 180,E1 -26652.308,E2 -26652.308} C_VEL
LIN {X 0,Y 247.138,Z 394.397,A -85,B 0,C 180,E1 -26653.789,E2 -26653.789} C_VEL
LIN {X 0,Y 247.157,Z 394.944,A -85,B 0,C 180,E1 -26654.495,E2 -26654.495} C_VEL
LIN {X 0,Y 242.447,Z 428.767,A -85,B 0,C 180,E1 -26655.135,E2 -26655.135} C_VEL
LIN {X 0,Y 238.499,Z 446.494,A -85,B 0,C 180,E1 -26655.524,E2 -26655.524} C_VEL
LIN {X 0,Y 233.078,Z 463.854,A -85,B 0,C 180,E1 -26656.033,E2 -26656.033} C_VEL
LIN {X 0,Y 227.356,Z 478.219,A -85,B 0,C 180,E1 -26656.615,E2 -26656.615} C_VEL
LIN {X 0,Y 220.015,Z 493.472,A -85,B 0,C 180,E1 -26657.392,E2 -26657.392} C_VEL
LIN {X 0,Y 212.013,Z 507.519,A -85,B 0,C 180,E1 -26658.402,E2 -26658.402} C_VEL
LIN {X 0,Y 202.467,Z 521.689,A -85,B 0,C 180,E1 -26659.689,E2 -26659.689} C_VEL
LIN {X 0,Y 192.293,Z 534.624,A -85,B 0,C 180,E1 -26661.257,E2 -26661.257} C_VEL
LIN {X 0,Y 181.597,Z 546.559,A -85,B 0,C 180,E1 -26663.201,E2 -26663.201} C_VEL
LIN {X 0,Y 172.62,Z 555.498,A -85,B 0,C 180,E1 -26665.062,E2 -26665.062} C_VEL
LIN {X 0,Y 162.456,Z 564.496,A -85,B 0,C 180,E1 -26667.523,E2 -26667.523} C_VEL
LIN {X 0,Y 151.178,Z 573.448,A -85,B 0,C 180,E1 -26670.755,E2 -26670.755} C_VEL
LIN {X 0,Y 140.73,Z 580.899,A -85,B 0,C 180,E1 -26674.515,E2 -26674.515} C_VEL
LIN {X 0,Y 130.907,Z 587.157,A -85,B 0,C 180,E1 -26678.882,E2 -26678.882} C_VEL
LIN {X 0,Y 123.066,Z 591.743,A -85,B 0,C 180,E1 -26683.258,E2 -26683.258} C_VEL
LIN {X 0,Y 116.089,Z 595.584,A -85,B 0,C 180,E1 -26688.248,E2 -26688.248} C_VEL
LIN {X 0,Y 109.288,Z 598.961,A -85,B 0,C 180,E1 -26694.638,E2 -26694.638} C_VEL
LIN {X 0,Y 104.763,Z 601.106,A -85,B 0,C 180,E1 -26700.562,E2 -26700.562} C_VEL
LIN {X 0,Y 102.294,Z 601.965,A -85,B 0,C 180,E1 -26703.492,E2 -26703.492} C_VEL
LIN {X 0,Y 97.107,Z 602.965,A -85,B 0,C 180,E1 -26708.314,E2 -26708.314} C_VEL
LIN {X 0,Y 93.306,Z 603.38,A -85,B 0,C 180,E1 -26712.518,E2 -26712.518} C_VEL
LIN {X 0,Y 91.508,Z 603.469,A -85,B 0,C 180,E1 -26716.022,E2 -26716.022} C_VEL
LIN {X 0,Y 91.231,Z 603.455,A -85,B 0,C 180,E1 -26717.249,E2 -26717.249} C_VEL
LIN {X 0,Y 90.798,Z 603.067,A -85,B 0,C 180,E1 -26725.562,E2 -26725.562} C_VEL
LIN {X 0,Y 90.971,Z 602.542,A -85,B 0,C 180,E1 -26730.001,E2 -26730.001} C_VEL
LIN {X 0,Y 90.823,Z 601.757,A -85,B 0,C 180,E1 -26734.439,E2 -26734.439} C_VEL
LIN {X 0,Y 91.353,Z 599.278,A -85,B 0,C 180,E1 -26743.345,E2 -26743.345} C_VEL
LIN {X 0,Y 93.569,Z 595.801,A -85,B 0,C 180,E1 -26752.059,E2 -26752.059} C_VEL
LIN {X 0,Y 97.431,Z 591.108,A -85,B 0,C 180,E1 -26760.328,E2 -26760.328} C_VEL
LIN {X 0,Y 102.989,Z 585.214,A -85,B 0,C 180,E1 -26767.892,E2 -26767.892} C_VEL
LIN {X 0,Y 110.052,Z 578.029,A -85,B 0,C 180,E1 -26774.626,E2 -26774.626} C_VEL
LIN {X 0,Y 118.396,Z 569.296,A -85,B 0,C 180,E1 -26780.506,E2 -26780.506} C_VEL
LIN {X 0,Y 126.593,Z 560.225,A -85,B 0,C 180,E1 -26784.972,E2 -26784.972} C_VEL
LIN {X 0,Y 135.338,Z 549.71,A -85,B 0,C 180,E1 -26788.899,E2 -26788.899} C_VEL
LIN {X 0,Y 143.409,Z 539.095,A -85,B 0,C 180,E1 -26791.899,E2 -26791.899} C_VEL
LIN {X 0,Y 151.838,Z 526.815,A -85,B 0,C 180,E1 -26794.5,E2 -26794.5} C_VEL
LIN {X 0,Y 159.761,Z 513.637,A -85,B 0,C 180,E1 -26796.677,E2 -26796.677} C_VEL
LIN {X 0,Y 167.178,Z 499.511,A -85,B 0,C 180,E1 -26798.452,E2 -26798.452} C_VEL
LIN {X 0,Y 173.945,Z 484.18,A -85,B 0,C 180,E1 -26799.948,E2 -26799.948} C_VEL
LIN {X 0,Y 180.085,Z 467.227,A -85,B 0,C 180,E1 -26801.152,E2 -26801.152} C_VEL
LIN {X 0,Y 184.562,Z 451.497,A -85,B 0,C 180,E1 -26801.951,E2 -26801.951} C_VEL
LIN {X 0,Y 188.116,Z 434.957,A -85,B 0,C 180,E1 -26802.532,E2 -26802.532} C_VEL
LIN {X 0,Y 190.917,Z 413.249,A -85,B 0,C 180,E1 -26803.158,E2 -26803.158} C_VEL
LIN {X 0,Y 196.02,Z 366.746,A -85,B 0,C 180,E1 -26804.295,E2 -26804.295} C_VEL
LIN {X 0,Y 193.066,Z 360.124,A -85,B 0,C 180,E1 -26806.916,E2 -26806.916} C_VEL
LIN {X 0,Y 189.665,Z 353.016,A -85,B 0,C 180,E1 -26810.358,E2 -26810.358} C_VEL
LIN {X 0,Y 186.14,Z 346.162,A -85,B 0,C 180,E1 -26814.589,E2 -26814.589} C_VEL
LIN {X 0,Y 184.37,Z 342.801,A -85,B 0,C 180,E1 -26817.195,E2 -26817.195} C_VEL
LIN {X 0,Y 182.728,Z 339.644,A -85,B 0,C 180,E1 -26820.092,E2 -26820.092} C_VEL
LIN {X 0,Y 181.088,Z 336.088,A -85,B 0,C 180,E1 -26824.033,E2 -26824.033} C_VEL
LIN {X 0,Y 179.675,Z 333.988,A -85,B 0,C 180,E1 -26829.581,E2 -26829.581} C_VEL
LIN {X 0,Y 179.555,Z 332.871,A -85,B 0,C 180,E1 -26831.895,E2 -26831.895} C_VEL
LIN {X 0,Y 179.513,Z 333.048,A -85,B 0,C 180,E1 -26833.961,E2 -26833.961} C_VEL
LIN {X 0,Y 181.207,Z 337.032,A -85,B 0,C 180,E1 -26843.038,E2 -26843.038} C_VEL
LIN {X 0,Y 183.296,Z 341.065,A -85,B 0,C 180,E1 -26847.584,E2 -26847.584} C_VEL
LIN {X 0,Y 185.597,Z 345.362,A -85,B 0,C 180,E1 -26851.205,E2 -26851.205} C_VEL
LIN {X 0,Y 188.527,Z 350.943,A -85,B 0,C 180,E1 -26854.931,E2 -26854.931} C_VEL
LIN {X 0,Y 192.104,Z 358.112,A -85,B 0,C 180,E1 -26858.695,E2 -26858.695} C_VEL
LIN {X 0,Y 195.85,Z 366.11,A -85,B 0,C 180,E1 -26862.056,E2 -26862.056} C_VEL
LIN {X 0,Y 189.502,Z 423.141,A -85,B 0,C 180,E1 -26863.505,E2 -26863.505} C_VEL
LIN {X 0,Y 186.553,Z 439.586,A -85,B 0,C 180,E1 -26864.067,E2 -26864.067} C_VEL
LIN {X 0,Y 182.367,Z 456.414,A -85,B 0,C 180,E1 -26864.917,E2 -26864.917} C_VEL
LIN {X 0,Y 177.438,Z 471.653,A -85,B 0,C 180,E1 -26865.923,E2 -26865.923} C_VEL
LIN {X 0,Y 171.488,Z 486.83,A -85,B 0,C 180,E1 -26867.292,E2 -26867.292} C_VEL
LIN {X 0,Y 164.566,Z 501.376,A -85,B 0,C 180,E1 -26868.958,E2 -26868.958} C_VEL
LIN {X 0,Y 157.36,Z 514.449,A -85,B 0,C 180,E1 -26870.887,E2 -26870.887} C_VEL
LIN {X 0,Y 149.253,Z 527.376,A -85,B 0,C 180,E1 -26873.345,E2 -26873.345} C_VEL
LIN {X 0,Y 140.17,Z 540.124,A -85,B 0,C 180,E1 -26876.527,E2 -26876.527} C_VEL
LIN {X 0,Y 131.161,Z 551.371,A -85,B 0,C 180,E1 -26880.287,E2 -26880.287} C_VEL
LIN {X 0,Y 122.756,Z 560.94,A -85,B 0,C 180,E1 -26884.571,E2 -26884.571} C_VEL
LIN {X 0,Y 113.975,Z 570.234,A -85,B 0,C 180,E1 -26890.174,E2 -26890.174} C_VEL
LIN {X 0,Y 106.335,Z 577.987,A -85,B 0,C 180,E1 -26896.624,E2 -26896.624} C_VEL
LIN {X 0,Y 100.074,Z 584.336,A -85,B 0,C 180,E1 -26903.952,E2 -26903.952} C_VEL
LIN {X 0,Y 95.252,Z 589.418,A -85,B 0,C 180,E1 -26912.113,E2 -26912.113} C_VEL
LIN {X 0,Y 92.533,Z 592.675,A -85,B 0,C 180,E1 -26919.119,E2 -26919.119} C_VEL
LIN {X 0,Y 90.647,Z 595.611,A -85,B 0,C 180,E1 -26928.065,E2 -26928.065} C_VEL
LIN {X 0,Y 90.191,Z 597.675,A -85,B 0,C 180,E1 -26937.873,E2 -26937.873} C_VEL
LIN {X 0,Y 91.425,Z 598.542,A -85,B 0,C 180,E1 -26947.948,E2 -26947.948} C_VEL
LIN {X 0,Y 94.877,Z 598.197,A -85,B 0,C 180,E1 -26958.189,E2 -26958.189} C_VEL
LIN {X 0,Y 100.309,Z 596.683,A -85,B 0,C 180,E1 -26967.218,E2 -26967.218} C_VEL
LIN {X 0,Y 108.045,Z 593.813,A -85,B 0,C 180,E1 -26975.592,E2 -26975.592} C_VEL
LIN {X 0,Y 117.722,Z 589.506,A -85,B 0,C 180,E1 -26982.779,E2 -26982.779} C_VEL
LIN {X 0,Y 128.955,Z 583.736,A -85,B 0,C 180,E1 -26988.803,E2 -26988.803} C_VEL
LIN {X 0,Y 141.378,Z 576.368,A -85,B 0,C 180,E1 -26993.817,E2 -26993.817} C_VEL
LIN {X 0,Y 152.541,Z 568.832,A -85,B 0,C 180,E1 -26997.359,E2 -26997.359} C_VEL
LIN {X 0,Y 163.454,Z 560.43,A -85,B 0,C 180,E1 -27000.251,E2 -27000.251} C_VEL
LIN {X 0,Y 173.942,Z 551.283,A -85,B 0,C 180,E1 -27002.579,E2 -27002.579} C_VEL
LIN {X 0,Y 184.921,Z 540.495,A -85,B 0,C 180,E1 -27004.684,E2 -27004.684} C_VEL
LIN {X 0,Y 195.418,Z 528.629,A -85,B 0,C 180,E1 -27006.437,E2 -27006.437} C_VEL
LIN {X 0,Y 205.799,Z 514.945,A -85,B 0,C 180,E1 -27007.978,E2 -27007.978} C_VEL
LIN {X 0,Y 215.178,Z 500.427,A -85,B 0,C 180,E1 -27009.202,E2 -27009.202} C_VEL
LIN {X 0,Y 222.896,Z 486.281,A -85,B 0,C 180,E1 -27010.142,E2 -27010.142} C_VEL
LIN {X 0,Y 229.465,Z 471.916,A -85,B 0,C 180,E1 -27010.893,E2 -27010.893} C_VEL
LIN {X 0,Y 235.344,Z 455.874,A -85,B 0,C 180,E1 -27011.522,E2 -27011.522} C_VEL
LIN {X 0,Y 239.425,Z 441.39,A -85,B 0,C 180,E1 -27011.933,E2 -27011.933} C_VEL
LIN {X 0,Y 242.969,Z 423.978,A -85,B 0,C 180,E1 -27012.305,E2 -27012.305} C_VEL
LIN {X 0,Y 246.195,Z 400.864,A -85,B 0,C 180,E1 -27012.721,E2 -27012.721} C_VEL
LIN {X 0,Y 246.192,Z 400.919,A -85,B 0,C 180,E1 -27012.924,E2 -27012.924} C_VEL
LIN {X 0,Y 242.054,Z 429.468,A -85,B 0,C 180,E1 -27013.467,E2 -27013.467} C_VEL
LIN {X 0,Y 238.156,Z 446.606,A -85,B 0,C 180,E1 -27013.825,E2 -27013.825} C_VEL
LIN {X 0,Y 232.698,Z 463.822,A -85,B 0,C 180,E1 -27014.283,E2 -27014.283} C_VEL
LIN {X 0,Y 227.137,Z 477.573,A -85,B 0,C 180,E1 -27014.781,E2 -27014.781} C_VEL
LIN {X 0,Y 219.704,Z 492.837,A -85,B 0,C 180,E1 -27015.5,E2 -27015.5} C_VEL
LIN {X 0,Y 211.549,Z 506.917,A -85,B 0,C 180,E1 -27016.413,E2 -27016.413} C_VEL
LIN {X 0,Y 201.836,Z 521.114,A -85,B 0,C 180,E1 -27017.602,E2 -27017.602} C_VEL
LIN {X 0,Y 191.296,Z 534.302,A -85,B 0,C 180,E1 -27019.077,E2 -27019.077} C_VEL
LIN {X 0,Y 180.474,Z 546.066,A -85,B 0,C 180,E1 -27020.839,E2 -27020.839} C_VEL
LIN {X 0,Y 169.759,Z 556.362,A -85,B 0,C 180,E1 -27022.909,E2 -27022.909} C_VEL
LIN {X 0,Y 157.853,Z 566.425,A -85,B 0,C 180,E1 -27025.637,E2 -27025.637} C_VEL
LIN {X 0,Y 147.401,Z 574.193,A -85,B 0,C 180,E1 -27028.476,E2 -27028.476} C_VEL
LIN {X 0,Y 136.824,Z 581.334,A -85,B 0,C 180,E1 -27032.059,E2 -27032.059} C_VEL
LIN {X 0,Y 124.115,Z 588.865,A -85,B 0,C 180,E1 -27037.559,E2 -27037.559} C_VEL
LIN {X 0,Y 114.95,Z 593.635,A -85,B 0,C 180,E1 -27042.807,E2 -27042.807} C_VEL
LIN {X 0,Y 106.984,Z 597.48,A -85,B 0,C 180,E1 -27048.937,E2 -27048.937} C_VEL
LIN {X 0,Y 97.903,Z 601.344,A -85,B 0,C 180,E1 -27059.477,E2 -27059.477} C_VEL
LIN {X 0,Y 93.597,Z 602.854,A -85,B 0,C 180,E1 -27067.95,E2 -27067.95} C_VEL
LIN {X 0,Y 91.231,Z 603.455,A -85,B 0,C 180,E1 -27077.249,E2 -27077.249} C_VEL
LIN {X 0,Y 90.157,Z 603.375,A -85,B 0,C 180,E1 -27080.924,E2 -27080.924} C_VEL
LIN {X 0,Y 88.384,Z 603.083,A -85,B 0,C 180,E1 -27084.571,E2 -27084.571} C_VEL
LIN {X 0,Y 83.952,Z 601.392,A -85,B 0,C 180,E1 -27094.834,E2 -27094.834} C_VEL
LIN {X 0,Y 83.735,Z 600.75,A -85,B 0,C 180,E1 -27097.556,E2 -27097.556} C_VEL
LIN {X 0,Y 84.382,Z 598.846,A -85,B 0,C 180,E1 -27104.471,E2 -27104.471} C_VEL
LIN {X 0,Y 87.855,Z 594.17,A -85,B 0,C 180,E1 -27116.103,E2 -27116.103} C_VEL
LIN {X 0,Y 92.659,Z 589.128,A -85,B 0,C 180,E1 -27124.672,E2 -27124.672} C_VEL
LIN {X 0,Y 99.147,Z 582.84,A -85,B 0,C 180,E1 -27132.331,E2 -27132.331} C_VEL
LIN {X 0,Y 107.942,Z 574.362,A -85,B 0,C 180,E1 -27139.515,E2 -27139.515} C_VEL
LIN {X 0,Y 116.351,Z 565.854,A -85,B 0,C 180,E1 -27144.632,E2 -27144.632} C_VEL
LIN {X 0,Y 125.142,Z 556.287,A -85,B 0,C 180,E1 -27148.92,E2 -27148.92} C_VEL
LIN {X 0,Y 134.536,Z 545.053,A -85,B 0,C 180,E1 -27152.631,E2 -27152.631} C_VEL
LIN {X 0,Y 144.469,Z 531.743,A -85,B 0,C 180,E1 -27155.802,E2 -27155.802} C_VEL
LIN {X 0,Y 152.819,Z 518.969,A -85,B 0,C 180,E1 -27158.057,E2 -27158.057} C_VEL
LIN {X 0,Y 160.832,Z 504.862,A -85,B 0,C 180,E1 -27159.968,E2 -27159.968} C_VEL
LIN {X 0,Y 167.729,Z 490.689,A -85,B 0,C 180,E1 -27161.443,E2 -27161.443} C_VEL
LIN {X 0,Y 173.95,Z 475.467,A -85,B 0,C 180,E1 -27162.651,E2 -27162.651} C_VEL
LIN {X 0,Y 179.447,Z 458.601,A -85,B 0,C 180,E1 -27163.644,E2 -27163.644} C_VEL
LIN {X 0,Y 183.63,Z 442.008,A -85,B 0,C 180,E1 -27164.288,E2 -27164.288} C_VEL
LIN {X 0,Y 186.474,Z 425.424,A -85,B 0,C 180,E1 -27164.784,E2 -27164.784} C_VEL
LIN {X 0,Y 192.735,Z 370.229,A -85,B 0,C 180,E1 -27166.121,E2 -27166.121} C_VEL
LIN {X 0,Y 188.802,Z 361.368,A -85,B 0,C 180,E1 -27170.074,E2 -27170.074} C_VEL
LIN {X 0,Y 185.211,Z 353.989,A -85,B 0,C 180,E1 -27174.405,E2 -27174.405} C_VEL
LIN {X 0,Y 182.903,Z 349.341,A -85,B 0,C 180,E1 -27177.904,E2 -27177.904} C_VEL
LIN {X 0,Y 181.389,Z 346.298,A -85,B 0,C 180,E1 -27180.787,E2 -27180.787} C_VEL
LIN {X 0,Y 179.948,Z 343.009,A -85,B 0,C 180,E1 -27184.48,E2 -27184.48} C_VEL
LIN {X 0,Y 178.664,Z 340.867,A -85,B 0,C 180,E1 -27190.043,E2 -27190.043} C_VEL
LIN {X 0,Y 178.594,Z 339.921,A -85,B 0,C 180,E1 -27192.018,E2 -27192.018} C_VEL
LIN {X 0,Y 178.537,Z 340.291,A -85,B 0,C 180,E1 -27194.227,E2 -27194.227} C_VEL
LIN {X 0,Y 180.065,Z 343.92,A -85,B 0,C 180,E1 -27202.604,E2 -27202.604} C_VEL
LIN {X 0,Y 182.184,Z 348.267,A -85,B 0,C 180,E1 -27207.416,E2 -27207.416} C_VEL
LIN {X 0,Y 184.231,Z 352.266,A -85,B 0,C 180,E1 -27210.74,E2 -27210.74} C_VEL
LIN {X 0,Y 186.867,Z 357.56,A -85,B 0,C 180,E1 -27214.275,E2 -27214.275} C_VEL
LIN {X 0,Y 190.099,Z 364.339,A -85,B 0,C 180,E1 -27217.854,E2 -27217.854} C_VEL
LIN {X 0,Y 192.54,Z 369.785,A -85,B 0,C 180,E1 -27220.226,E2 -27220.226} C_VEL
LIN {X 0,Y 186.572,Z 422.291,A -85,B 0,C 180,E1 -27221.524,E2 -27221.524} C_VEL
LIN {X 0,Y 183.483,Z 439.535,A -85,B 0,C 180,E1 -27222.087,E2 -27222.087} C_VEL
LIN {X 0,Y 179.266,Z 456.228,A -85,B 0,C 180,E1 -27222.892,E2 -27222.892} C_VEL
LIN {X 0,Y 174.281,Z 471.43,A -85,B 0,C 180,E1 -27223.852,E2 -27223.852} C_VEL
LIN {X 0,Y 168.202,Z 486.601,A -85,B 0,C 180,E1 -27225.163,E2 -27225.163} C_VEL
LIN {X 0,Y 160.667,Z 502.097,A -85,B 0,C 180,E1 -27226.884,E2 -27226.884} C_VEL
LIN {X 0,Y 153.272,Z 515.082,A -85,B 0,C 180,E1 -27228.766,E2 -27228.766} C_VEL
LIN {X 0,Y 144.315,Z 528.786,A -85,B 0,C 180,E1 -27231.353,E2 -27231.353} C_VEL
LIN {X 0,Y 135.511,Z 540.648,A -85,B 0,C 180,E1 -27234.305,E2 -27234.305} C_VEL
LIN {X 0,Y 126.188,Z 551.865,A -85,B 0,C 180,E1 -27238.055,E2 -27238.055} C_VEL
LIN {X 0,Y 117.406,Z 561.393,A -85,B 0,C 180,E1 -27242.359,E2 -27242.359} C_VEL
LIN {X 0,Y 108.194,Z 570.647,A -85,B 0,C 180,E1 -27248.067,E2 -27248.067} C_VEL
LIN {X 0,Y 101.038,Z 577.512,A -85,B 0,C 180,E1 -27253.844,E2 -27253.844} C_VEL
LIN {X 0,Y 94.22,Z 583.943,A -85,B 0,C 180,E1 -27261.419,E2 -27261.419} C_VEL
LIN {X 0,Y 88.879,Z 589.171,A -85,B 0,C 180,E1 -27269.999,E2 -27269.999} C_VEL
LIN {X 0,Y 85.186,Z 593.287,A -85,B 0,C 180,E1 -27279.496,E2 -27279.496} C_VEL
LIN {X 0,Y 83.343,Z 596.196,A -85,B 0,C 180,E1 -27289.711,E2 -27289.711} C_VEL
LIN {X 0,Y 83.227,Z 598.06,A -85,B 0,C 180,E1 -27300.44,E2 -27300.44} C_VEL
LIN {X 0,Y 85.096,Z 598.825,A -85,B 0,C 180,E1 -27311.352,E2 -27311.352} C_VEL
LIN {X 0,Y 89.314,Z 598.302,A -85,B 0,C 180,E1 -27321.892,E2 -27321.892} C_VEL
LIN {X 0,Y 95.95,Z 596.539,A -85,B 0,C 180,E1 -27331.513,E2 -27331.513} C_VEL
LIN {X 0,Y 104.798,Z 593.476,A -85,B 0,C 180,E1 -27339.857,E2 -27339.857} C_VEL
LIN {X 0,Y 115.49,Z 589.026,A -85,B 0,C 180,E1 -27346.813,E2 -27346.813} C_VEL
LIN {X 0,Y 127.577,Z 583.056,A -85,B 0,C 180,E1 -27352.55,E2 -27352.55} C_VEL
LIN {X 0,Y 140.718,Z 575.471,A -85,B 0,C 180,E1 -27357.247,E2 -27357.247} C_VEL
LIN {X 0,Y 152.137,Z 567.85,A -85,B 0,C 180,E1 -27360.464,E2 -27360.464} C_VEL
LIN {X 0,Y 163.648,Z 559.172,A -85,B 0,C 180,E1 -27363.176,E2 -27363.176} C_VEL
LIN {X 0,Y 176.563,Z 547.926,A -85,B 0,C 180,E1 -27365.681,E2 -27365.681} C_VEL
LIN {X 0,Y 188.823,Z 535.434,A -85,B 0,C 180,E1 -27367.711,E2 -27367.711} C_VEL
LIN {X 0,Y 199.349,Z 522.959,A -85,B 0,C 180,E1 -27369.21,E2 -27369.21} C_VEL
LIN {X 0,Y 208.069,Z 511.063,A -85,B 0,C 180,E1 -27370.347,E2 -27370.347} C_VEL
LIN {X 0,Y 217.21,Z 496.523,A -85,B 0,C 180,E1 -27371.39,E2 -27371.39} C_VEL
LIN {X 0,Y 225.288,Z 481.085,A -85,B 0,C 180,E1 -27372.259,E2 -27372.259} C_VEL
LIN {X 0,Y 227.448,Z 476.258,A -85,B 0,C 180,E1 -27372.491,E2 -27372.491} C_VEL
LIN {X 0,Y 226.698,Z 477.979,A -85,B 0,C 180,E1 -27372.995,E2 -27372.995} C_VEL
LIN {X 0,Y 219.632,Z 492.298,A -85,B 0,C 180,E1 -27373.603,E2 -27373.603} C_VEL
LIN {X 0,Y 211.347,Z 506.45,A -85,B 0,C 180,E1 -27374.424,E2 -27374.424} C_VEL
LIN {X 0,Y 201.492,Z 520.613,A -85,B 0,C 180,E1 -27375.522,E2 -27375.522} C_VEL
LIN {X 0,Y 190.904,Z 533.615,A -85,B 0,C 180,E1 -27376.834,E2 -27376.834} C_VEL
LIN {X 0,Y 180.018,Z 545.29,A -85,B 0,C 180,E1 -27378.445,E2 -27378.445} C_VEL
LIN {X 0,Y 168.694,Z 555.945,A -85,B 0,C 180,E1 -27380.388,E2 -27380.388} C_VEL
LIN {X 0,Y 156.43,Z 565.978,A -85,B 0,C 180,E1 -27382.929,E2 -27382.929} C_VEL
LIN {X 0,Y 143.803,Z 574.995,A -85,B 0,C 180,E1 -27386.094,E2 -27386.094} C_VEL
LIN {X 0,Y 133.179,Z 581.761,A -85,B 0,C 180,E1 -27389.46,E2 -27389.46} C_VEL
LIN {X 0,Y 122.437,Z 587.77,A -85,B 0,C 180,E1 -27393.666,E2 -27393.666} C_VEL
LIN {X 0,Y 112.74,Z 592.649,A -85,B 0,C 180,E1 -27398.563,E2 -27398.563} C_VEL
LIN {X 0,Y 101.666,Z 597.561,A -85,B 0,C 180,E1 -27406.27,E2 -27406.27} C_VEL
LIN {X 0,Y 94.549,Z 600.282,A -85,B 0,C 180,E1 -27413.514,E2 -27413.514} C_VEL
LIN {X 0,Y 89.054,Z 602.178,A -85,B 0,C 180,E1 -27421.74,E2 -27421.74} C_VEL
LIN {X 0,Y 85.384,Z 603.075,A -85,B 0,C 180,E1 -27430.779,E2 -27430.779} C_VEL
LIN {X 0,Y 83.826,Z 603.144,A -85,B 0,C 180,E1 -27440.349,E2 -27440.349} C_VEL
LIN {X 0,Y 83.875,Z 602.215,A -85,B 0,C 180,E1 -27450.001,E2 -27450.001} C_VEL
LIN {X 0,Y 83.735,Z 600.75,A -85,B 0,C 180,E1 -27457.556,E2 -27457.556} C_VEL
LIN {X 0,Y 83.349,Z 599.741,A -85,B 0,C 180,E1 -27461.531,E2 -27461.531} C_VEL
LIN {X 0,Y 81.592,Z 597.644,A -85,B 0,C 180,E1 -27468.156,E2 -27468.156} C_VEL
LIN {X 0,Y 80.697,Z 595.673,A -85,B 0,C 180,E1 -27473.586,E2 -27473.586} C_VEL
LIN {X 0,Y 81.209,Z 593.95,A -85,B 0,C 180,E1 -27477.606,E2 -27477.606} C_VEL
LIN {X 0,Y 81.713,Z 593.341,A -85,B 0,C 180,E1 -27478.887,E2 -27478.887} C_VEL
LIN {X 0,Y 86.805,Z 588.447,A -85,B 0,C 180,E1 -27487.39,E2 -27487.39} C_VEL
LIN {X 0,Y 93.923,Z 582.068,A -85,B 0,C 180,E1 -27495.306,E2 -27495.306} C_VEL
LIN {X 0,Y 103.021,Z 573.791,A -85,B 0,C 180,E1 -27502.347,E2 -27502.347} C_VEL
LIN {X 0,Y 112.324,Z 564.817,A -85,B 0,C 180,E1 -27507.639,E2 -27507.639} C_VEL
LIN {X 0,Y 121.457,Z 555.172,A -85,B 0,C 180,E1 -27511.816,E2 -27511.816} C_VEL
LIN {X 0,Y 131.357,Z 543.653,A -85,B 0,C 180,E1 -27515.444,E2 -27515.444} C_VEL
LIN {X 0,Y 140.908,Z 531.206,A -85,B 0,C 180,E1 -27518.272,E2 -27518.272} C_VEL
LIN {X 0,Y 150.027,Z 517.507,A -85,B 0,C 180,E1 -27520.581,E2 -27520.581} C_VEL
LIN {X 0,Y 157.716,Z 504.169,A -85,B 0,C 180,E1 -27522.268,E2 -27522.268} C_VEL
LIN {X 0,Y 164.777,Z 489.884,A -85,B 0,C 180,E1 -27523.67,E2 -27523.67} C_VEL
LIN {X 0,Y 171.125,Z 474.517,A -85,B 0,C 180,E1 -27524.824,E2 -27524.824} C_VEL
LIN {X 0,Y 176.742,Z 457.511,A -85,B 0,C 180,E1 -27525.754,E2 -27525.754} C_VEL
LIN {X 0,Y 180.956,Z 440.753,A -85,B 0,C 180,E1 -27526.357,E2 -27526.357} C_VEL
LIN {X 0,Y 183.657,Z 424.908,A -85,B 0,C 180,E1 -27526.804,E2 -27526.804} C_VEL
LIN {X 0,Y 189.577,Z 373.977,A -85,B 0,C 180,E1 -27527.991,E2 -27527.991} C_VEL
LIN {X 0,Y 186.097,Z 365.822,A -85,B 0,C 180,E1 -27531.876,E2 -27531.876} C_VEL
LIN {X 0,Y 183.061,Z 359.225,A -85,B 0,C 180,E1 -27536.02,E2 -27536.02} C_VEL
LIN {X 0,Y 181.182,Z 355.343,A -85,B 0,C 180,E1 -27539.14,E2 -27539.14} C_VEL
LIN {X 0,Y 180.083,Z 352.955,A -85,B 0,C 180,E1 -27541.479,E2 -27541.479} C_VEL
LIN {X 0,Y 178.795,Z 349.9,A -85,B 0,C 180,E1 -27545.007,E2 -27545.007} C_VEL
LIN {X 0,Y 177.641,Z 347.554,A -85,B 0,C 180,E1 -27550.936,E2 -27550.936} C_VEL
LIN {X 0,Y 177.586,Z 347.263,A -85,B 0,C 180,E1 -27553.926,E2 -27553.926} C_VEL
LIN {X 0,Y 178.923,Z 350.777,A -85,B 0,C 180,E1 -27562.13,E2 -27562.13} C_VEL
LIN {X 0,Y 180.794,Z 354.828,A -85,B 0,C 180,E1 -27566.683,E2 -27566.683} C_VEL
LIN {X 0,Y 182.689,Z 358.787,A -85,B 0,C 180,E1 -27570.007,E2 -27570.007} C_VEL
LIN {X 0,Y 185.388,Z 364.511,A -85,B 0,C 180,E1 -27573.807,E2 -27573.807} C_VEL
LIN {X 0,Y 188.409,Z 371.177,A -85,B 0,C 180,E1 -27577.292,E2 -27577.292} C_VEL
LIN {X 0,Y 189.403,Z 373.543,A -85,B 0,C 180,E1 -27578.346,E2 -27578.346} C_VEL
LIN {X 0,Y 183.644,Z 422.858,A -85,B 0,C 180,E1 -27579.528,E2 -27579.528} C_VEL
LIN {X 0,Y 180.497,Z 439.924,A -85,B 0,C 180,E1 -27580.062,E2 -27580.062} C_VEL
LIN {X 0,Y 176.382,Z 455.922,A -85,B 0,C 180,E1 -27580.794,E2 -27580.794} C_VEL
LIN {X 0,Y 171.256,Z 471.346,A -85,B 0,C 180,E1 -27581.722,E2 -27581.722} C_VEL
LIN {X 0,Y 164.751,Z 487.212,A -85,B 0,C 180,E1 -27583.042,E2 -27583.042} C_VEL
LIN {X 0,Y 156.982,Z 502.726,A -85,B 0,C 180,E1 -27584.706,E2 -27584.706} C_VEL
LIN {X 0,Y 149.396,Z 515.635,A -85,B 0,C 180,E1 -27586.528,E2 -27586.528} C_VEL
LIN {X 0,Y 140.47,Z 528.875,A -85,B 0,C 180,E1 -27588.953,E2 -27588.953} C_VEL
LIN {X 0,Y 131.08,Z 541.098,A -85,B 0,C 180,E1 -27591.932,E2 -27591.932} C_VEL
LIN {X 0,Y 121.414,Z 552.293,A -85,B 0,C 180,E1 -27595.641,E2 -27595.641} C_VEL
LIN {X 0,Y 112.241,Z 561.787,A -85,B 0,C 180,E1 -27599.938,E2 -27599.938} C_VEL
LIN {X 0,Y 102.575,Z 571.006,A -85,B 0,C 180,E1 -27605.725,E2 -27605.725} C_VEL
LIN {X 0,Y 94.027,Z 578.692,A -85,B 0,C 180,E1 -27612.603,E2 -27612.603} C_VEL
LIN {X 0,Y 86.918,Z 585.012,A -85,B 0,C 180,E1 -27620.692,E2 -27620.692} C_VEL
LIN {X 0,Y 81.423,Z 590.031,A -85,B 0,C 180,E1 -27629.999,E2 -27629.999} C_VEL
LIN {X 0,Y 77.71,Z 593.957,A -85,B 0,C 180,E1 -27640.419,E2 -27640.419} C_VEL
LIN {X 0,Y 76.105,Z 596.773,A -85,B 0,C 180,E1 -27651.676,E2 -27651.676} C_VEL
LIN {X 0,Y 76.509,Z 598.521,A -85,B 0,C 180,E1 -27664.236,E2 -27664.236} C_VEL
LIN {X 0,Y 79.054,Z 599.014,A -85,B 0,C 180,E1 -27675.33,E2 -27675.33} C_VEL
LIN {X 0,Y 84.362,Z 598.382,A -85,B 0,C 180,E1 -27686.413,E2 -27686.413} C_VEL
LIN {X 0,Y 92.175,Z 596.408,A -85,B 0,C 180,E1 -27696.195,E2 -27696.195} C_VEL
LIN {X 0,Y 102.157,Z 593.122,A -85,B 0,C 180,E1 -27704.389,E2 -27704.389} C_VEL
LIN {X 0,Y 113.841,Z 588.473,A -85,B 0,C 180,E1 -27711.015,E2 -27711.015} C_VEL
LIN {X 0,Y 123.429,Z 583.998,A -85,B 0,C 180,E1 -27715.146,E2 -27715.146} C_VEL
LIN {X 0,Y 135.832,Z 577.33,A -85,B 0,C 180,E1 -27719.35,E2 -27719.35} C_VEL
LIN {X 0,Y 148.517,Z 569.473,A -85,B 0,C 180,E1 -27722.712,E2 -27722.712} C_VEL
LIN {X 0,Y 160.375,Z 560.946,A -85,B 0,C 180,E1 -27725.329,E2 -27725.329} C_VEL
LIN {X 0,Y 171.671,Z 551.641,A -85,B 0,C 180,E1 -27727.383,E2 -27727.383} C_VEL
LIN {X 0,Y 182.791,Z 541.278,A -85,B 0,C 180,E1 -27729.145,E2 -27729.145} C_VEL
LIN {X 0,Y 193.995,Z 529.184,A -85,B 0,C 180,E1 -27730.688,E2 -27730.688} C_VEL
LIN {X 0,Y 204.761,Z 515.575,A -85,B 0,C 180,E1 -27731.991,E2 -27731.991} C_VEL
LIN {X 0,Y 208.684,Z 509.993,A -85,B 0,C 180,E1 -27732.411,E2 -27732.411} C_VEL
LIN {X 0,Y 208.911,Z 509.674,A -85,B 0,C 180,E1 -27732.692,E2 -27732.692} C_VEL
LIN {X 0,Y 198.919,Z 523.371,A -85,B 0,C 180,E1 -27733.693,E2 -27733.693} C_VEL
LIN {X 0,Y 189.013,Z 535.088,A -85,B 0,C 180,E1 -27734.822,E2 -27734.822} C_VEL
LIN {X 0,Y 178.042,Z 546.338,A -85,B 0,C 180,E1 -27736.292,E2 -27736.292} C_VEL
LIN {X 0,Y 166.377,Z 556.842,A -85,B 0,C 180,E1 -27738.12,E2 -27738.12} C_VEL
LIN {X 0,Y 153.819,Z 566.765,A -85,B 0,C 180,E1 -27740.509,E2 -27740.509} C_VEL
LIN {X 0,Y 140.543,Z 575.777,A -85,B 0,C 180,E1 -27743.581,E2 -27743.581} C_VEL
LIN {X 0,Y 126.945,Z 583.759,A -85,B 0,C 180,E1 -27747.653,E2 -27747.653} C_VEL
LIN {X 0,Y 115.939,Z 589.409,A -85,B 0,C 180,E1 -27751.938,E2 -27751.938} C_VEL
LIN {X 0,Y 105.738,Z 593.994,A -85,B 0,C 180,E1 -27757.102,E2 -27757.102} C_VEL
LIN {X 0,Y 96.593,Z 597.613,A -85,B 0,C 180,E1 -27763.318,E2 -27763.318} C_VEL
LIN {X 0,Y 88.875,Z 600.275,A -85,B 0,C 180,E1 -27770.759,E2 -27770.759} C_VEL
LIN {X 0,Y 82.804,Z 602.062,A -85,B 0,C 180,E1 -27779.388,E2 -27779.388} C_VEL
LIN {X 0,Y 78.643,Z 602.894,A -85,B 0,C 180,E1 -27789.057,E2 -27789.057} C_VEL
LIN {X 0,Y 76.801,Z 602.902,A -85,B 0,C 180,E1 -27799.456,E2 -27799.456} C_VEL
LIN {X 0,Y 76.771,Z 601.876,A -85,B 0,C 180,E1 -27810.002,E2 -27810.002} C_VEL
LIN {X 0,Y 76.83,Z 599.865,A -85,B 0,C 180,E1 -27820.543,E2 -27820.543} C_VEL
LIN {X 0,Y 78.631,Z 596.679,A -85,B 0,C 180,E1 -27830.949,E2 -27830.949} C_VEL
LIN {X 0,Y 81.713,Z 593.341,A -85,B 0,C 180,E1 -27838.887,E2 -27838.887} C_VEL
LIN {X 0,Y 82.992,Z 591.442,A -85,B 0,C 180,E1 -27842.677,E2 -27842.677} C_VEL
LIN {X 0,Y 85.399,Z 585.007,A -85,B 0,C 180,E1 -27853.934,E2 -27853.934} C_VEL
LIN {X 0,Y 87.498,Z 582.549,A -85,B 0,C 180,E1 -27857.222,E2 -27857.222} C_VEL
LIN {X 0,Y 88.486,Z 581.654,A -85,B 0,C 180,E1 -27858.185,E2 -27858.185} C_VEL
LIN {X 0,Y 98.194,Z 573.371,A -85,B 0,C 180,E1 -27865.331,E2 -27865.331} C_VEL
LIN {X 0,Y 108.611,Z 563.768,A -85,B 0,C 180,E1 -27870.876,E2 -27870.876} C_VEL
LIN {X 0,Y 118.005,Z 554.151,A -85,B 0,C 180,E1 -27874.854,E2 -27874.854} C_VEL
LIN {X 0,Y 127.021,Z 544.057,A -85,B 0,C 180,E1 -27877.936,E2 -27877.936} C_VEL
LIN {X 0,Y 137.623,Z 530.66,A -85,B 0,C 180,E1 -27880.863,E2 -27880.863} C_VEL
LIN {X 0,Y 146.935,Z 516.968,A -85,B 0,C 180,E1 -27883.06,E2 -27883.06} C_VEL
LIN {X 0,Y 154.868,Z 503.481,A -85,B 0,C 180,E1 -27884.652,E2 -27884.652} C_VEL
LIN {X 0,Y 162.083,Z 489.08,A -85,B 0,C 180,E1 -27885.975,E2 -27885.975} C_VEL
LIN {X 0,Y 168.552,Z 473.534,A -85,B 0,C 180,E1 -27887.071,E2 -27887.071} C_VEL
LIN {X 0,Y 173.869,Z 457.742,A -85,B 0,C 180,E1 -27887.874,E2 -27887.874} C_VEL
LIN {X 0,Y 178.213,Z 440.841,A -85,B 0,C 180,E1 -27888.446,E2 -27888.446} C_VEL
LIN {X 0,Y 180.986,Z 425.068,A -85,B 0,C 180,E1 -27888.864,E2 -27888.864} C_VEL
LIN {X 0,Y 186.589,Z 377.755,A -85,B 0,C 180,E1 -27889.959,E2 -27889.959} C_VEL
LIN {X 0,Y 183.942,Z 371.364,A -85,B 0,C 180,E1 -27893.18,E2 -27893.18} C_VEL
LIN {X 0,Y 181.165,Z 364.969,A -85,B 0,C 180,E1 -27897.339,E2 -27897.339} C_VEL
LIN {X 0,Y 179.007,Z 360.009,A -85,B 0,C 180,E1 -27901.679,E2 -27901.679} C_VEL
LIN {X 0,Y 177.659,Z 356.78,A -85,B 0,C 180,E1 -27905.541,E2 -27905.541} C_VEL
LIN {X 0,Y 176.668,Z 354.379,A -85,B 0,C 180,E1 -27911.473,E2 -27911.473} C_VEL
LIN {X 0,Y 176.61,Z 354.549,A -85,B 0,C 180,E1 -27914.386,E2 -27914.386} C_VEL
LIN {X 0,Y 177.826,Z 357.765,A -85,B 0,C 180,E1 -27921.779,E2 -27921.779} C_VEL
LIN {X 0,Y 179.496,Z 361.569,A -85,B 0,C 180,E1 -27926.087,E2 -27926.087} C_VEL
LIN {X 0,Y 181.39,Z 365.746,A -85,B 0,C 180,E1 -27929.608,E2 -27929.608} C_VEL
LIN {X 0,Y 183.729,Z 371.044,A -85,B 0,C 180,E1 -27933.079,E2 -27933.079} C_VEL
LIN {X 0,Y 186.409,Z 377.288,A -85,B 0,C 180,E1 -27936.354,E2 -27936.354} C_VEL
LIN {X 0,Y 186.278,Z 379.405,A -85,B 0,C 180,E1 -27936.498,E2 -27936.498} C_VEL
LIN {X 0,Y 180.642,Z 425.631,A -85,B 0,C 180,E1 -27937.527,E2 -27937.527} C_VEL
LIN {X 0,Y 177.145,Z 442.993,A -85,B 0,C 180,E1 -27938.068,E2 -27938.068} C_VEL
LIN {X 0,Y 172.531,Z 459.51,A -85,B 0,C 180,E1 -27938.826,E2 -27938.826} C_VEL
LIN {X 0,Y 166.965,Z 475.102,A -85,B 0,C 180,E1 -27939.808,E2 -27939.808} C_VEL
LIN {X 0,Y 160.767,Z 489.382,A -85,B 0,C 180,E1 -27940.975,E2 -27940.975} C_VEL
LIN {X 0,Y 153.53,Z 503.357,A -85,B 0,C 180,E1 -27942.427,E2 -27942.427} C_VEL
LIN {X 0,Y 145.008,Z 517.377,A -85,B 0,C 180,E1 -27944.366,E2 -27944.366} C_VEL
LIN {X 0,Y 135.843,Z 530.367,A -85,B 0,C 180,E1 -27946.724,E2 -27946.724} C_VEL
LIN {X 0,Y 125.411,Z 543.234,A -85,B 0,C 180,E1 -27949.874,E2 -27949.874} C_VEL
LIN {X 0,Y 115.444,Z 554.137,A -85,B 0,C 180,E1 -27953.589,E2 -27953.589} C_VEL
LIN {X 0,Y 105.969,Z 563.462,A -85,B 0,C 180,E1 -27957.955,E2 -27957.955} C_VEL
LIN {X 0,Y 95.937,Z 572.419,A -85,B 0,C 180,E1 -27963.925,E2 -27963.925} C_VEL
LIN {X 0,Y 87.047,Z 579.866,A -85,B 0,C 180,E1 -27971.157,E2 -27971.157} C_VEL
LIN {X 0,Y 79.62,Z 586.001,A -85,B 0,C 180,E1 -27979.83,E2 -27979.83} C_VEL
LIN {X 0,Y 73.924,Z 590.899,A -85,B 0,C 180,E1 -27989.998,E2 -27989.998} C_VEL
LIN {X 0,Y 70.242,Z 594.626,A -85,B 0,C 180,E1 -28001.542,E2 -28001.542} C_VEL
LIN {X 0,Y 68.83,Z 597.3,A -85,B 0,C 180,E1 -28014.104,E2 -28014.104} C_VEL
LIN {X 0,Y 69.626,Z 598.741,A -85,B 0,C 180,E1 -28026.146,E2 -28026.146} C_VEL
LIN {X 0,Y 72.349,Z 599.25,A -85,B 0,C 180,E1 -28037.158,E2 -28037.158} C_VEL
LIN {X 0,Y 76.798,Z 598.877,A -85,B 0,C 180,E1 -28046.696,E2 -28046.696} C_VEL
LIN {X 0,Y 84.224,Z 597.495,A -85,B 0,C 180,E1 -28056.614,E2 -28056.614} C_VEL
LIN {X 0,Y 94.412,Z 594.709,A -85,B 0,C 180,E1 -28065.394,E2 -28065.394} C_VEL
LIN {X 0,Y 106.437,Z 590.514,A -85,B 0,C 180,E1 -28072.411,E2 -28072.411} C_VEL
LIN {X 0,Y 119.552,Z 584.952,A -85,B 0,C 180,E1 -28077.911,E2 -28077.911} C_VEL
LIN {X 0,Y 133.634,Z 577.825,A -85,B 0,C 180,E1 -28082.278,E2 -28082.278} C_VEL
LIN {X 0,Y 147.014,Z 569.832,A -85,B 0,C 180,E1 -28085.486,E2 -28085.486} C_VEL
LIN {X 0,Y 159.976,Z 560.78,A -85,B 0,C 180,E1 -28088.042,E2 -28088.042} C_VEL
LIN {X 0,Y 173.127,Z 550.082,A -85,B 0,C 180,E1 -28090.136,E2 -28090.136} C_VEL
LIN {X 0,Y 185.036,Z 538.805,A -85,B 0,C 180,E1 -28091.78,E2 -28091.78} C_VEL
LIN {X 0,Y 188.937,Z 534.771,A -85,B 0,C 180,E1 -28092.256,E2 -28092.256} C_VEL
LIN {X 0,Y 187.358,Z 536.488,A -85,B 0,C 180,E1 -28092.77,E2 -28092.77} C_VEL
LIN {X 0,Y 175.259,Z 548.449,A -85,B 0,C 180,E1 -28094.227,E2 -28094.227} C_VEL
LIN {X 0,Y 164.327,Z 557.803,A -85,B 0,C 180,E1 -28095.791,E2 -28095.791} C_VEL
LIN {X 0,Y 151.483,Z 567.483,A -85,B 0,C 180,E1 -28097.998,E2 -28097.998} C_VEL
LIN {X 0,Y 139.769,Z 575.187,A -85,B 0,C 180,E1 -28100.423,E2 -28100.423} C_VEL
LIN {X 0,Y 126.774,Z 582.623,A -85,B 0,C 180,E1 -28103.839,E2 -28103.839} C_VEL
LIN {X 0,Y 115.116,Z 588.449,A -85,B 0,C 180,E1 -28107.722,E2 -28107.722} C_VEL
LIN {X 0,Y 101.567,Z 594.2,A -85,B 0,C 180,E1 -28113.869,E2 -28113.869} C_VEL
LIN {X 0,Y 87.418,Z 599.113,A -85,B 0,C 180,E1 -28123.654,E2 -28123.654} C_VEL
LIN {X 0,Y 78.645,Z 601.496,A -85,B 0,C 180,E1 -28133.54,E2 -28133.54} C_VEL
LIN {X 0,Y 74.085,Z 602.474,A -85,B 0,C 180,E1 -28141.687,E2 -28141.687} C_VEL
LIN {X 0,Y 70.59,Z 602.763,A -85,B 0,C 180,E1 -28152.623,E2 -28152.623} C_VEL
LIN {X 0,Y 69.518,Z 602.214,A -85,B 0,C 180,E1 -28164.199,E2 -28164.199} C_VEL
LIN {X 0,Y 69.689,Z 601.539,A -85,B 0,C 180,E1 -28170.002,E2 -28170.002} C_VEL
LIN {X 0,Y 69.799,Z 599.421,A -85,B 0,C 180,E1 -28181.619,E2 -28181.619} C_VEL
LIN {X 0,Y 71.978,Z 596.172,A -85,B 0,C 180,E1 -28192.991,E2 -28192.991} C_VEL
LIN {X 0,Y 76.5,Z 591.822,A -85,B 0,C 180,E1 -28203.452,E2 -28203.452} C_VEL
LIN {X 0,Y 82.973,Z 586.289,A -85,B 0,C 180,E1 -28212.659,E2 -28212.659} C_VEL
LIN {X 0,Y 88.486,Z 581.654,A -85,B 0,C 180,E1 -28218.185,E2 -28218.185} C_VEL
LIN {X 0,Y 91.186,Z 578.995,A -85,B 0,C 180,E1 -28221.079,E2 -28221.079} C_VEL
LIN {X 0,Y 94.505,Z 574.362,A -85,B 0,C 180,E1 -28226.1,E2 -28226.1} C_VEL
LIN {X 0,Y 98.317,Z 569.312,A -85,B 0,C 180,E1 -28230.648,E2 -28230.648} C_VEL
LIN {X 0,Y 101.614,Z 565.988,A -85,B 0,C 180,E1 -28232.717,E2 -28232.717} C_VEL
LIN {X 0,Y 112.455,Z 555.641,A -85,B 0,C 180,E1 -28237.194,E2 -28237.194} C_VEL
LIN {X 0,Y 122.944,Z 544.393,A -85,B 0,C 180,E1 -28240.599,E2 -28240.599} C_VEL
LIN {X 0,Y 132.258,Z 533.067,A -85,B 0,C 180,E1 -28243.038,E2 -28243.038} C_VEL
LIN {X 0,Y 141.792,Z 519.902,A -85,B 0,C 180,E1 -28245.134,E2 -28245.134} C_VEL
LIN {X 0,Y 150.015,Z 506.745,A -85,B 0,C 180,E1 -28246.733,E2 -28246.733} C_VEL
LIN {X 0,Y 158.015,Z 491.719,A -85,B 0,C 180,E1 -28248.095,E2 -28248.095} C_VEL
LIN {X 0,Y 165.012,Z 475.692,A -85,B 0,C 180,E1 -28249.188,E2 -28249.188} C_VEL
LIN {X 0,Y 170.398,Z 460.336,A -85,B 0,C 180,E1 -28249.968,E2 -28249.968} C_VEL
LIN {X 0,Y 174.803,Z 444.52,A -85,B 0,C 180,E1 -28250.498,E2 -28250.498} C_VEL
LIN {X 0,Y 177.945,Z 429.092,A -85,B 0,C 180,E1 -28250.888,E2 -28250.888} C_VEL
LIN {X 0,Y 183.761,Z 381.649,A -85,B 0,C 180,E1 -28251.951,E2 -28251.951} C_VEL
LIN {X 0,Y 181.753,Z 376.578,A -85,B 0,C 180,E1 -28254.716,E2 -28254.716} C_VEL
LIN {X 0,Y 179.476,Z 370.988,A -85,B 0,C 180,E1 -28258.476,E2 -28258.476} C_VEL
LIN {X 0,Y 177.682,Z 366.621,A -85,B 0,C 180,E1 -28262.437,E2 -28262.437} C_VEL
LIN {X 0,Y 176.61,Z 363.763,A -85,B 0,C 180,E1 -28265.82,E2 -28265.82} C_VEL
LIN {X 0,Y 175.699,Z 361.488,A -85,B 0,C 180,E1 -28271.537,E2 -28271.537} C_VEL
LIN {X 0,Y 175.651,Z 361.604,A -85,B 0,C 180,E1 -28274.274,E2 -28274.274} C_VEL
LIN {X 0,Y 176.726,Z 364.692,A -85,B 0,C 180,E1 -28281.379,E2 -28281.379} C_VEL
LIN {X 0,Y 178.245,Z 368.372,A -85,B 0,C 180,E1 -28285.545,E2 -28285.545} C_VEL
LIN {X 0,Y 179.902,Z 372.286,A -85,B 0,C 180,E1 -28288.871,E2 -28288.871} C_VEL
LIN {X 0,Y 182.168,Z 377.722,A -85,B 0,C 180,E1 -28292.433,E2 -28292.433} C_VEL
LIN {X 0,Y 183.663,Z 381.573,A -85,B 0,C 180,E1 -28294.47,E2 -28294.47} C_VEL
LIN {X 0,Y 178.044,Z 426.435,A -85,B 0,C 180,E1 -28295.417,E2 -28295.417} C_VEL
LIN {X 0,Y 174.391,Z 444.117,A -85,B 0,C 180,E1 -28295.955,E2 -28295.955} C_VEL
LIN {X 0,Y 169.733,Z 460.238,A -85,B 0,C 180,E1 -28296.655,E2 -28296.655} C_VEL
LIN {X 0,Y 164.054,Z 475.721,A -85,B 0,C 180,E1 -28297.577,E2 -28297.577} C_VEL
LIN {X 0,Y 157.047,Z 491.268,A -85,B 0,C 180,E1 -28298.793,E2 -28298.793} C_VEL
LIN {X 0,Y 149.537,Z 505.23,A -85,B 0,C 180,E1 -28300.206,E2 -28300.206} C_VEL
LIN {X 0,Y 140.807,Z 519.051,A -85,B 0,C 180,E1 -28302.059,E2 -28302.059} C_VEL
LIN {X 0,Y 131.567,Z 531.598,A -85,B 0,C 180,E1 -28304.29,E2 -28304.29} C_VEL
LIN {X 0,Y 121.43,Z 543.632,A -85,B 0,C 180,E1 -28307.151,E2 -28307.151} C_VEL
LIN {X 0,Y 111.094,Z 554.508,A -85,B 0,C 180,E1 -28310.756,E2 -28310.756} C_VEL
LIN {X 0,Y 101.214,Z 563.82,A -85,B 0,C 180,E1 -28315.049,E2 -28315.049} C_VEL
LIN {X 0,Y 90.665,Z 572.75,A -85,B 0,C 180,E1 -28321.021,E2 -28321.021} C_VEL
LIN {X 0,Y 82.313,Z 579.331,A -85,B 0,C 180,E1 -28327.404,E2 -28327.404} C_VEL
LIN {X 0,Y 74.155,Z 585.621,A -85,B 0,C 180,E1 -28336.293,E2 -28336.293} C_VEL
LIN {X 0,Y 67.733,Z 590.602,A -85,B 0,C 180,E1 -28347.024,E2 -28347.024} C_VEL
LIN {X 0,Y 63.863,Z 594.091,A -85,B 0,C 180,E1 -28357.93,E2 -28357.93} C_VEL
LIN {X 0,Y 61.718,Z 597.422,A -85,B 0,C 180,E1 -28374.359,E2 -28374.359} C_VEL
LIN {X 0,Y 62.817,Z 598.956,A -85,B 0,C 180,E1 -28388.449,E2 -28388.449} C_VEL
LIN {X 0,Y 66.139,Z 599.469,A -85,B 0,C 180,E1 -28400.39,E2 -28400.39} C_VEL
LIN {X 0,Y 71.962,Z 599.027,A -85,B 0,C 180,E1 -28411.513,E2 -28411.513} C_VEL
LIN {X 0,Y 81.216,Z 597.383,A -85,B 0,C 180,E1 -28422.145,E2 -28422.145} C_VEL
LIN {X 0,Y 92.618,Z 594.454,A -85,B 0,C 180,E1 -28430.547,E2 -28430.547} C_VEL
LIN {X 0,Y 105.564,Z 590.131,A -85,B 0,C 180,E1 -28436.97,E2 -28436.97} C_VEL
LIN {X 0,Y 116.187,Z 585.838,A -85,B 0,C 180,E1 -28440.918,E2 -28440.918} C_VEL
LIN {X 0,Y 130.509,Z 579.023,A -85,B 0,C 180,E1 -28444.989,E2 -28444.989} C_VEL
LIN {X 0,Y 143.814,Z 571.49,A -85,B 0,C 180,E1 -28447.912,E2 -28447.912} C_VEL
LIN {X 0,Y 157.152,Z 562.635,A -85,B 0,C 180,E1 -28450.316,E2 -28450.316} C_VEL
LIN {X 0,Y 168.781,Z 553.75,A -85,B 0,C 180,E1 -28452.017,E2 -28452.017} C_VEL
LIN {X 0,Y 167.497,Z 554.875,A -85,B 0,C 180,E1 -28452.759,E2 -28452.759} C_VEL
LIN {X 0,Y 154.339,Z 564.899,A -85,B 0,C 180,E1 -28454.621,E2 -28454.621} C_VEL
LIN {X 0,Y 142.978,Z 572.462,A -85,B 0,C 180,E1 -28456.568,E2 -28456.568} C_VEL
LIN {X 0,Y 130.278,Z 579.858,A -85,B 0,C 180,E1 -28459.26,E2 -28459.26} C_VEL
LIN {X 0,Y 117.953,Z 586.046,A -85,B 0,C 180,E1 -28462.556,E2 -28462.556} C_VEL
LIN {X 0,Y 106.159,Z 591.208,A -85,B 0,C 180,E1 -28466.657,E2 -28466.657} C_VEL
LIN {X 0,Y 92.428,Z 596.183,A -85,B 0,C 180,E1 -28473.24,E2 -28473.24} C_VEL
LIN {X 0,Y 82.616,Z 599.123,A -85,B 0,C 180,E1 -28480.042,E2 -28480.042} C_VEL
LIN {X 0,Y 72.477,Z 601.543,A -85,B 0,C 180,E1 -28490.872,E2 -28490.872} C_VEL
LIN {X 0,Y 65.462,Z 602.535,A -85,B 0,C 180,E1 -28504.57,E2 -28504.57} C_VEL
LIN {X 0,Y 62.794,Z 602.324,A -85,B 0,C 180,E1 -28517.067,E2 -28517.067} C_VEL
LIN {X 0,Y 62.426,Z 601.916,A -85,B 0,C 180,E1 -28523.538,E2 -28523.538} C_VEL
LIN {X 0,Y 62.596,Z 601.195,A -85,B 0,C 180,E1 -28530.002,E2 -28530.002} C_VEL
LIN {X 0,Y 62.814,Z 598.964,A -85,B 0,C 180,E1 -28542.932,E2 -28542.932} C_VEL
LIN {X 0,Y 65.44,Z 595.658,A -85,B 0,C 180,E1 -28555.443,E2 -28555.443} C_VEL
LIN {X 0,Y 70.574,Z 591.183,A -85,B 0,C 180,E1 -28566.692,E2 -28566.692} C_VEL
LIN {X 0,Y 77.815,Z 585.555,A -85,B 0,C 180,E1 -28576.266,E2 -28576.266} C_VEL
LIN {X 0,Y 86.727,Z 578.539,A -85,B 0,C 180,E1 -28584.132,E2 -28584.132} C_VEL
LIN {X 0,Y 96.949,Z 570.065,A -85,B 0,C 180,E1 -28590.448,E2 -28590.448} C_VEL
LIN {X 0,Y 101.614,Z 565.988,A -85,B 0,C 180,E1 -28592.717,E2 -28592.717} C_VEL
LIN {X 0,Y 104.947,Z 562.628,A -85,B 0,C 180,E1 -28594.633,E2 -28594.633} C_VEL
LIN {X 0,Y 112.81,Z 551.942,A -85,B 0,C 180,E1 -28600.975,E2 -28600.975} C_VEL
LIN {X 0,Y 116.021,Z 548.051,A -85,B 0,C 180,E1 -28602.533,E2 -28602.533} C_VEL
LIN {X 0,Y 117.253,Z 546.692,A -85,B 0,C 180,E1 -28602.912,E2 -28602.912} C_VEL
LIN {X 0,Y 127.102,Z 535.417,A -85,B 0,C 180,E1 -28605.386,E2 -28605.386} C_VEL
LIN {X 0,Y 136.82,Z 522.747,A -85,B 0,C 180,E1 -28607.413,E2 -28607.413} C_VEL
LIN {X 0,Y 145.379,Z 509.769,A -85,B 0,C 180,E1 -28608.929,E2 -28608.929} C_VEL
LIN {X 0,Y 153.336,Z 495.631,A -85,B 0,C 180,E1 -28610.208,E2 -28610.208} C_VEL
LIN {X 0,Y 160.441,Z 480.602,A -85,B 0,C 180,E1 -28611.239,E2 -28611.239} C_VEL
LIN {X 0,Y 166.341,Z 465.514,A -85,B 0,C 180,E1 -28611.991,E2 -28611.991} C_VEL
LIN {X 0,Y 171.101,Z 450.027,A -85,B 0,C 180,E1 -28612.534,E2 -28612.534} C_VEL
LIN {X 0,Y 174.908,Z 433.375,A -85,B 0,C 180,E1 -28612.948,E2 -28612.948} C_VEL
LIN {X 0,Y 177.953,Z 411.991,A -85,B 0,C 180,E1 -28613.433,E2 -28613.433} C_VEL
LIN {X 0,Y 181.166,Z 385.658,A -85,B 0,C 180,E1 -28613.961,E2 -28613.961} C_VEL
LIN {X 0,Y 178.62,Z 378.992,A -85,B 0,C 180,E1 -28618.123,E2 -28618.123} C_VEL
LIN {X 0,Y 176.749,Z 374.019,A -85,B 0,C 180,E1 -28622.279,E2 -28622.279} C_VEL
LIN {X 0,Y 175.49,Z 370.671,A -85,B 0,C 180,E1 -28626.379,E2 -28626.379} C_VEL
LIN {X 0,Y 174.734,Z 368.58,A -85,B 0,C 180,E1 -28631.602,E2 -28631.602} C_VEL
LIN {X 0,Y 174.68,Z 368.784,A -85,B 0,C 180,E1 -28634.355,E2 -28634.355} C_VEL
LIN {X 0,Y 175.624,Z 371.569,A -85,B 0,C 180,E1 -28640.921,E2 -28640.921} C_VEL
LIN {X 0,Y 176.988,Z 375.101,A -85,B 0,C 180,E1 -28644.961,E2 -28644.961} C_VEL
LIN {X 0,Y 178.756,Z 379.571,A -85,B 0,C 180,E1 -28648.694,E2 -28648.694} C_VEL
LIN {X 0,Y 181.038,Z 385.483,A -85,B 0,C 180,E1 -28652.393,E2 -28652.393} C_VEL
LIN {X 0,Y 175.78,Z 426.674,A -85,B 0,C 180,E1 -28653.235,E2 -28653.235} C_VEL
LIN {X 0,Y 172.089,Z 444.26,A -85,B 0,C 180,E1 -28653.735,E2 -28653.735} C_VEL
LIN {X 0,Y 167.181,Z 460.94,A -85,B 0,C 180,E1 -28654.411,E2 -28654.411} C_VEL
LIN {X 0,Y 161.396,Z 476.31,A -85,B 0,C 180,E1 -28655.267,E2 -28655.267} C_VEL
LIN {X 0,Y 154.083,Z 492.125,A -85,B 0,C 180,E1 -28656.433,E2 -28656.433} C_VEL
LIN {X 0,Y 145.762,Z 507.013,A -85,B 0,C 180,E1 -28657.858,E2 -28657.858} C_VEL
LIN {X 0,Y 136.839,Z 520.615,A -85,B 0,C 180,E1 -28659.61,E2 -28659.61} C_VEL
LIN {X 0,Y 126.643,Z 533.909,A -85,B 0,C 180,E1 -28661.898,E2 -28661.898} C_VEL
LIN {X 0,Y 116.237,Z 545.659,A -85,B 0,C 180,E1 -28664.729,E2 -28664.729} C_VEL
LIN {X 0,Y 105.548,Z 556.247,A -85,B 0,C 180,E1 -28668.251,E2 -28668.251} C_VEL
LIN {X 0,Y 93.879,Z 566.487,A -85,B 0,C 180,E1 -28673.208,E2 -28673.208} C_VEL
LIN {X 0,Y 83.019,Z 575.046,A -85,B 0,C 180,E1 -28679.472,E2 -28679.472} C_VEL
LIN {X 0,Y 73.284,Z 582.15,A -85,B 0,C 180,E1 -28687.442,E2 -28687.442} C_VEL
LIN {X 0,Y 64.593,Z 588.234,A -85,B 0,C 180,E1 -28698.304,E2 -28698.304} C_VEL
LIN {X 0,Y 58.901,Z 592.453,A -85,B 0,C 180,E1 -28709.998,E2 -28709.998} C_VEL
LIN {X 0,Y 56.694,Z 594.394,A -85,B 0,C 180,E1 -28717.381,E2 -28717.381} C_VEL
LIN {X 0,Y 54.651,Z 597.221,A -85,B 0,C 180,E1 -28732.69,E2 -28732.69} C_VEL
LIN {X 0,Y 55.723,Z 599.006,A -85,B 0,C 180,E1 -28749.092,E2 -28749.092} C_VEL
LIN {X 0,Y 60.321,Z 599.686,A -85,B 0,C 180,E1 -28764.639,E2 -28764.639} C_VEL
LIN {X 0,Y 68.327,Z 599.12,A -85,B 0,C 180,E1 -28777.772,E2 -28777.772} C_VEL
LIN {X 0,Y 79.01,Z 597.273,A -85,B 0,C 180,E1 -28788.075,E2 -28788.075} C_VEL
LIN {X 0,Y 91.601,Z 594.154,A -85,B 0,C 180,E1 -28795.845,E2 -28795.845} C_VEL
LIN {X 0,Y 105.458,Z 589.688,A -85,B 0,C 180,E1 -28801.616,E2 -28801.616} C_VEL
LIN {X 0,Y 120.136,Z 583.758,A -85,B 0,C 180,E1 -28806.025,E2 -28806.025} C_VEL
LIN {X 0,Y 135.35,Z 576.236,A -85,B 0,C 180,E1 -28809.41,E2 -28809.41} C_VEL
LIN {X 0,Y 148.985,Z 568.174,A -85,B 0,C 180,E1 -28811.819,E2 -28811.819} C_VEL
LIN {X 0,Y 150.956,Z 566.924,A -85,B 0,C 180,E1 -28812.133,E2 -28812.133} C_VEL
LIN {X 0,Y 151.05,Z 566.871,A -85,B 0,C 180,E1 -28812.298,E2 -28812.298} C_VEL
LIN {X 0,Y 137.843,Z 575.099,A -85,B 0,C 180,E1 -28814.374,E2 -28814.374} C_VEL
LIN {X 0,Y 124.905,Z 582,A -85,B 0,C 180,E1 -28816.96,E2 -28816.96} C_VEL
LIN {X 0,Y 112.294,Z 587.826,A -85,B 0,C 180,E1 -28820.157,E2 -28820.157} C_VEL
LIN {X 0,Y 100.16,Z 592.533,A -85,B 0,C 180,E1 -28824.196,E2 -28824.196} C_VEL
LIN {X 0,Y 88.688,Z 596.342,A -85,B 0,C 180,E1 -28829.349,E2 -28829.349} C_VEL
LIN {X 0,Y 73.423,Z 600.244,A -85,B 0,C 180,E1 -28840.029,E2 -28840.029} C_VEL
LIN {X 0,Y 65.147,Z 601.702,A -85,B 0,C 180,E1 -28849.667,E2 -28849.667} C_VEL
LIN {X 0,Y 59.076,Z 602.356,A -85,B 0,C 180,E1 -28861.587,E2 -28861.587} C_VEL
LIN {X 0,Y 55.849,Z 602.03,A -85,B 0,C 180,E1 -28875.425,E2 -28875.425} C_VEL
LIN {X 0,Y 55.491,Z 600.846,A -85,B 0,C 180,E1 -28890.002,E2 -28890.002} C_VEL
LIN {X 0,Y 55.85,Z 598.493,A -85,B 0,C 180,E1 -28904.579,E2 -28904.579} C_VEL
LIN {X 0,Y 59.05,Z 595.126,A -85,B 0,C 180,E1 -28918.431,E2 -28918.431} C_VEL
LIN {X 0,Y 65.358,Z 590.207,A -85,B 0,C 180,E1 -28931.174,E2 -28931.174} C_VEL
LIN {X 0,Y 72.983,Z 584.752,A -85,B 0,C 180,E1 -28940.389,E2 -28940.389} C_VEL
LIN {X 0,Y 82.691,Z 577.666,A -85,B 0,C 180,E1 -28948.204,E2 -28948.204} C_VEL
LIN {X 0,Y 93.594,Z 569.037,A -85,B 0,C 180,E1 -28954.302,E2 -28954.302} C_VEL
LIN {X 0,Y 103.821,Z 560.116,A -85,B 0,C 180,E1 -28958.559,E2 -28958.559} C_VEL
LIN {X 0,Y 114.436,Z 549.709,A -85,B 0,C 180,E1 -28962.117,E2 -28962.117} C_VEL
LIN {X 0,Y 117.253,Z 546.692,A -85,B 0,C 180,E1 -28962.912,E2 -28962.912} C_VEL
LIN {X 0,Y 120.677,Z 542.664,A -85,B 0,C 180,E1 -28964.146,E2 -28964.146} C_VEL
LIN {X 0,Y 129.831,Z 528.759,A -85,B 0,C 180,E1 -28969.056,E2 -28969.056} C_VEL
LIN {X 0,Y 133.026,Z 524.163,A -85,B 0,C 180,E1 -28969.978,E2 -28969.978} C_VEL
LIN {X 0,Y 142.308,Z 510.566,A -85,B 0,C 180,E1 -28971.48,E2 -28971.48} C_VEL
LIN {X 0,Y 150.578,Z 496.323,A -85,B 0,C 180,E1 -28972.663,E2 -28972.663} C_VEL
LIN {X 0,Y 157.792,Z 481.495,A -85,B 0,C 180,E1 -28973.611,E2 -28973.611} C_VEL
LIN {X 0,Y 164.202,Z 465.423,A -85,B 0,C 180,E1 -28974.339,E2 -28974.339} C_VEL
LIN {X 0,Y 169.142,Z 449.575,A -85,B 0,C 180,E1 -28974.823,E2 -28974.823} C_VEL
LIN {X 0,Y 172.978,Z 432.88,A -85,B 0,C 180,E1 -28975.194,E2 -28975.194} C_VEL
LIN {X 0,Y 176.203,Z 410.284,A -85,B 0,C 180,E1 -28975.669,E2 -28975.669} C_VEL
LIN {X 0,Y 178.714,Z 389.904,A -85,B 0,C 180,E1 -28976.076,E2 -28976.076} C_VEL
LIN {X 0,Y 176.705,Z 384.204,A -85,B 0,C 180,E1 -28979.89,E2 -28979.89} C_VEL
LIN {X 0,Y 175.209,Z 380.013,A -85,B 0,C 180,E1 -28983.742,E2 -28983.742} C_VEL
LIN {X 0,Y 174.395,Z 377.519,A -85,B 0,C 180,E1 -28986.944,E2 -28986.944} C_VEL
LIN {X 0,Y 173.767,Z 375.68,A -85,B 0,C 180,E1 -28991.667,E2 -28991.667} C_VEL
LIN {X 0,Y 173.727,Z 375.755,A -85,B 0,C 180,E1 -28994.047,E2 -28994.047} C_VEL
LIN {X 0,Y 174.536,Z 378.498,A -85,B 0,C 180,E1 -29000.491,E2 -29000.491} C_VEL
LIN {X 0,Y 175.689,Z 381.748,A -85,B 0,C 180,E1 -29004.259,E2 -29004.259} C_VEL
LIN {X 0,Y 177.078,Z 385.521,A -85,B 0,C 180,E1 -29007.489,E2 -29007.489} C_VEL
LIN {X 0,Y 178.622,Z 389.84,A -85,B 0,C 180,E1 -29010.336,E2 -29010.336} C_VEL
LIN {X 0,Y 173.792,Z 426.697,A -85,B 0,C 180,E1 -29011.005,E2 -29011.005} C_VEL
LIN {X 0,Y 170.152,Z 443.84,A -85,B 0,C 180,E1 -29011.44,E2 -29011.44} C_VEL
LIN {X 0,Y 165.312,Z 460.272,A -85,B 0,C 180,E1 -29012.047,E2 -29012.047} C_VEL
LIN {X 0,Y 159.42,Z 475.855,A -85,B 0,C 180,E1 -29012.821,E2 -29012.821} C_VEL
LIN {X 0,Y 152.303,Z 491.181,A -85,B 0,C 180,E1 -29013.839,E2 -29013.839} C_VEL
LIN {X 0,Y 144.766,Z 504.787,A -85,B 0,C 180,E1 -29014.991,E2 -29014.991} C_VEL
LIN {X 0,Y 135.632,Z 518.699,A -85,B 0,C 180,E1 -29016.567,E2 -29016.567} C_VEL
LIN {X 0,Y 125.763,Z 531.572,A -85,B 0,C 180,E1 -29018.522,E2 -29018.522} C_VEL
LIN {X 0,Y 116.008,Z 542.663,A -85,B 0,C 180,E1 -29020.775,E2 -29020.775} C_VEL
LIN {X 0,Y 104.909,Z 553.769,A -85,B 0,C 180,E1 -29023.932,E2 -29023.932} C_VEL
LIN {X 0,Y 92.599,Z 564.466,A -85,B 0,C 180,E1 -29028.386,E2 -29028.386} C_VEL
LIN {X 0,Y 80.934,Z 573.363,A -85,B 0,C 180,E1 -29034.115,E2 -29034.115} C_VEL
LIN {X 0,Y 71.496,Z 579.903,A -85,B 0,C 180,E1 -29040.56,E2 -29040.56} C_VEL
LIN {X 0,Y 61.98,Z 586.166,A -85,B 0,C 180,E1 -29050.111,E2 -29050.111} C_VEL
LIN {X 0,Y 54.302,Z 591.126,A -85,B 0,C 180,E1 -29062.562,E2 -29062.562} C_VEL
LIN {X 0,Y 49.185,Z 594.978,A -85,B 0,C 180,E1 -29078.213,E2 -29078.213} C_VEL
LIN {X 0,Y 47.532,Z 597.769,A -85,B 0,C 180,E1 -29096.329,E2 -29096.329} C_VEL
LIN {X 0,Y 49.646,Z 599.386,A -85,B 0,C 180,E1 -29115.053,E2 -29115.053} C_VEL
LIN {X 0,Y 55.878,Z 599.877,A -85,B 0,C 180,E1 -29131.686,E2 -29131.686} C_VEL
LIN {X 0,Y 65.579,Z 599.185,A -85,B 0,C 180,E1 -29144.681,E2 -29144.681} C_VEL
LIN {X 0,Y 78.71,Z 596.995,A -85,B 0,C 180,E1 -29154.877,E2 -29154.877} C_VEL
LIN {X 0,Y 94.971,Z 592.876,A -85,B 0,C 180,E1 -29162.575,E2 -29162.575} C_VEL
LIN {X 0,Y 110.092,Z 587.741,A -85,B 0,C 180,E1 -29167.335,E2 -29167.335} C_VEL
LIN {X 0,Y 125.2,Z 581.337,A -85,B 0,C 180,E1 -29170.79,E2 -29170.79} C_VEL
LIN {X 0,Y 131.055,Z 578.496,A -85,B 0,C 180,E1 -29171.868,E2 -29171.868} C_VEL
LIN {X 0,Y 129.605,Z 579.285,A -85,B 0,C 180,E1 -29172.567,E2 -29172.567} C_VEL
LIN {X 0,Y 116.481,Z 585.472,A -85,B 0,C 180,E1 -29175.127,E2 -29175.127} C_VEL
LIN {X 0,Y 103.684,Z 590.625,A -85,B 0,C 180,E1 -29178.391,E2 -29178.391} C_VEL
LIN {X 0,Y 90.869,Z 594.857,A -85,B 0,C 180,E1 -29182.75,E2 -29182.75} C_VEL
LIN {X 0,Y 79.671,Z 597.931,A -85,B 0,C 180,E1 -29188.104,E2 -29188.104} C_VEL
LIN {X 0,Y 64.218,Z 601.037,A -85,B 0,C 180,E1 -29200.001,E2 -29200.001} C_VEL
LIN {X 0,Y 52.866,Z 602.13,A -85,B 0,C 180,E1 -29217.878,E2 -29217.878} C_VEL
LIN {X 0,Y 48.955,Z 601.731,A -85,B 0,C 180,E1 -29233.317,E2 -29233.317} C_VEL
LIN {X 0,Y 48.373,Z 600.487,A -85,B 0,C 180,E1 -29250.002,E2 -29250.002} C_VEL
LIN {X 0,Y 48.956,Z 598.024,A -85,B 0,C 180,E1 -29266.687,E2 -29266.687} C_VEL
LIN {X 0,Y 52.835,Z 594.546,A -85,B 0,C 180,E1 -29282.147,E2 -29282.147} C_VEL
LIN {X 0,Y 59.609,Z 589.856,A -85,B 0,C 180,E1 -29295.026,E2 -29295.026} C_VEL
LIN {X 0,Y 68.599,Z 583.952,A -85,B 0,C 180,E1 -29305.046,E2 -29305.046} C_VEL
LIN {X 0,Y 79.114,Z 576.748,A -85,B 0,C 180,E1 -29312.667,E2 -29312.667} C_VEL
LIN {X 0,Y 90.692,Z 568.01,A -85,B 0,C 180,E1 -29318.423,E2 -29318.423} C_VEL
LIN {X 0,Y 101.384,Z 558.905,A -85,B 0,C 180,E1 -29322.395,E2 -29322.395} C_VEL
LIN {X 0,Y 113.04,Z 547.65,A -85,B 0,C 180,E1 -29325.805,E2 -29325.805} C_VEL
LIN {X 0,Y 123.824,Z 535.773,A -85,B 0,C 180,E1 -29328.26,E2 -29328.26} C_VEL
LIN {X 0,Y 133.026,Z 524.163,A -85,B 0,C 180,E1 -29329.978,E2 -29329.978} C_VEL
LIN {X 0,Y 136.15,Z 519.562,A -85,B 0,C 180,E1 -29330.83,E2 -29330.83} C_VEL
LIN {X 0,Y 140.378,Z 511.855,A -85,B 0,C 180,E1 -29332.731,E2 -29332.731} C_VEL
LIN {X 0,Y 144.368,Z 503.868,A -85,B 0,C 180,E1 -29334.47,E2 -29334.47} C_VEL
LIN {X 0,Y 147.036,Z 498.829,A -85,B 0,C 180,E1 -29335.087,E2 -29335.087} C_VEL
LIN {X 0,Y 154.993,Z 483.158,A -85,B 0,C 180,E1 -29336.004,E2 -29336.004} C_VEL
LIN {X 0,Y 161.48,Z 467.408,A -85,B 0,C 180,E1 -29336.655,E2 -29336.655} C_VEL
LIN {X 0,Y 166.686,Z 451.437,A -85,B 0,C 180,E1 -29337.123,E2 -29337.123} C_VEL
LIN {X 0,Y 170.932,Z 433.899,A -85,B 0,C 180,E1 -29337.456,E2 -29337.456} C_VEL
LIN {X 0,Y 174.011,Z 413.542,A -85,B 0,C 180,E1 -29337.859,E2 -29337.859} C_VEL
LIN {X 0,Y 176.437,Z 394.17,A -85,B 0,C 180,E1 -29338.227,E2 -29338.227} C_VEL
LIN {X 0,Y 174.856,Z 389.259,A -85,B 0,C 180,E1 -29341.906,E2 -29341.906} C_VEL
LIN {X 0,Y 173.887,Z 386.407,A -85,B 0,C 180,E1 -29344.812,E2 -29344.812} C_VEL
LIN {X 0,Y 173.35,Z 384.442,A -85,B 0,C 180,E1 -29347.34,E2 -29347.34} C_VEL
LIN {X 0,Y 172.807,Z 382.73,A -85,B 0,C 180,E1 -29351.733,E2 -29351.733} C_VEL
LIN {X 0,Y 172.751,Z 383.075,A -85,B 0,C 180,E1 -29354.526,E2 -29354.526} C_VEL
LIN {X 0,Y 173.448,Z 385.344,A -85,B 0,C 180,E1 -29359.981,E2 -29359.981} C_VEL
LIN {X 0,Y 174.585,Z 388.869,A -85,B 0,C 180,E1 -29364.016,E2 -29364.016} C_VEL
LIN {X 0,Y 176.089,Z 393.376,A -85,B 0,C 180,E1 -29367.635,E2 -29367.635} C_VEL
LIN {X 0,Y 176.351,Z 394.058,A -85,B 0,C 180,E1 -29368.152,E2 -29368.152} C_VEL
LIN {X 0,Y 171.977,Z 426.907,A -85,B 0,C 180,E1 -29368.735,E2 -29368.735} C_VEL
LIN {X 0,Y 168.207,Z 444.373,A -85,B 0,C 180,E1 -29369.132,E2 -29369.132} C_VEL
LIN {X 0,Y 163.303,Z 460.703,A -85,B 0,C 180,E1 -29369.68,E2 -29369.68} C_VEL
LIN {X 0,Y 157.318,Z 476.239,A -85,B 0,C 180,E1 -29370.371,E2 -29370.371} C_VEL
LIN {X 0,Y 150.089,Z 491.525,A -85,B 0,C 180,E1 -29371.288,E2 -29371.288} C_VEL
LIN {X 0,Y 141.575,Z 506.432,A -85,B 0,C 180,E1 -29372.444,E2 -29372.444} C_VEL
LIN {X 0,Y 132.282,Z 520.192,A -85,B 0,C 180,E1 -29373.886,E2 -29373.886} C_VEL
LIN {X 0,Y 121.34,Z 533.881,A -85,B 0,C 180,E1 -29375.818,E2 -29375.818} C_VEL
LIN {X 0,Y 109.757,Z 546.292,A -85,B 0,C 180,E1 -29378.335,E2 -29378.335} C_VEL
LIN {X 0,Y 98.369,Z 556.839,A -85,B 0,C 180,E1 -29381.393,E2 -29381.393} C_VEL
LIN {X 0,Y 85.707,Z 567.054,A -85,B 0,C 180,E1 -29385.812,E2 -29385.812} C_VEL
LIN {X 0,Y 73.659,Z 575.586,A -85,B 0,C 180,E1 -29391.669,E2 -29391.669} C_VEL
LIN {X 0,Y 62.524,Z 582.674,A -85,B 0,C 180,E1 -29399.613,E2 -29399.613} C_VEL
LIN {X 0,Y 51.619,Z 589.104,A -85,B 0,C 180,E1 -29412.373,E2 -29412.373} C_VEL
LIN {X 0,Y 46.864,Z 591.936,A -85,B 0,C 180,E1 -29421.373,E2 -29421.373} C_VEL
LIN {X 0,Y 41.595,Z 595.612,A -85,B 0,C 180,E1 -29439.724,E2 -29439.724} C_VEL
LIN {X 0,Y 40.552,Z 598.24,A -85,B 0,C 180,E1 -29461.323,E2 -29461.323} C_VEL
LIN {X 0,Y 44.205,Z 599.769,A -85,B 0,C 180,E1 -29482.643,E2 -29482.643} C_VEL
LIN {X 0,Y 52.409,Z 600.071,A -85,B 0,C 180,E1 -29499.825,E2 -29499.825} C_VEL
LIN {X 0,Y 63.856,Z 599.19,A -85,B 0,C 180,E1 -29512.095,E2 -29512.095} C_VEL
LIN {X 0,Y 77.309,Z 597.077,A -85,B 0,C 180,E1 -29520.579,E2 -29520.579} C_VEL
LIN {X 0,Y 91.948,Z 593.599,A -85,B 0,C 180,E1 -29526.479,E2 -29526.479} C_VEL
LIN {X 0,Y 107.294,Z 588.76,A -85,B 0,C 180,E1 -29530.734,E2 -29530.734} C_VEL
LIN {X 0,Y 111.886,Z 587.107,A -85,B 0,C 180,E1 -29531.727,E2 -29531.727} C_VEL
LIN {X 0,Y 108.203,Z 588.534,A -85,B 0,C 180,E1 -29533.032,E2 -29533.032} C_VEL
LIN {X 0,Y 95.193,Z 593.045,A -85,B 0,C 180,E1 -29536.313,E2 -29536.313} C_VEL
LIN {X 0,Y 82.6,Z 596.57,A -85,B 0,C 180,E1 -29540.628,E2 -29540.628} C_VEL
LIN {X 0,Y 70.679,Z 599.186,A -85,B 0,C 180,E1 -29546.507,E2 -29546.507} C_VEL
LIN {X 0,Y 59.84,Z 600.942,A -85,B 0,C 180,E1 -29554.707,E2 -29554.707} C_VEL
LIN {X 0,Y 50.633,Z 601.775,A -85,B 0,C 180,E1 -29566.055,E2 -29566.055} C_VEL
LIN {X 0,Y 44.044,Z 601.808,A -85,B 0,C 180,E1 -29581.403,E2 -29581.403} C_VEL
LIN {X 0,Y 41.238,Z 600.854,A -85,B 0,C 180,E1 -29600.19,E2 -29600.19} C_VEL
LIN {X 0,Y 41.275,Z 600.068,A -85,B 0,C 180,E1 -29610.003,E2 -29610.003} C_VEL
LIN {X 0,Y 41.246,Z 598.959,A -85,B 0,C 180,E1 -29619.813,E2 -29619.813} C_VEL
LIN {X 0,Y 44.037,Z 595.857,A -85,B 0,C 180,E1 -29638.608,E2 -29638.608} C_VEL
LIN {X 0,Y 50.528,Z 591.719,A -85,B 0,C 180,E1 -29654.066,E2 -29654.066} C_VEL
LIN {X 0,Y 59.526,Z 586.294,A -85,B 0,C 180,E1 -29665.739,E2 -29665.739} C_VEL
LIN {X 0,Y 70.26,Z 579.607,A -85,B 0,C 180,E1 -29674.194,E2 -29674.194} C_VEL
LIN {X 0,Y 82.075,Z 571.518,A -85,B 0,C 180,E1 -29680.378,E2 -29680.378} C_VEL
LIN {X 0,Y 94.613,Z 561.809,A -85,B 0,C 180,E1 -29684.942,E2 -29684.942} C_VEL
LIN {X 0,Y 105.923,Z 551.643,A -85,B 0,C 180,E1 -29688.146,E2 -29688.146} C_VEL
LIN {X 0,Y 117.524,Z 539.76,A -85,B 0,C 180,E1 -29690.65,E2 -29690.65} C_VEL
LIN {X 0,Y 128.475,Z 526.777,A -85,B 0,C 180,E1 -29692.522,E2 -29692.522} C_VEL
LIN {X 0,Y 138.179,Z 513.268,A -85,B 0,C 180,E1 -29693.996,E2 -29693.996} C_VEL
LIN {X 0,Y 147.036,Z 498.829,A -85,B 0,C 180,E1 -29695.087,E2 -29695.087} C_VEL
LIN {X 0,Y 149.601,Z 493.721,A -85,B 0,C 180,E1 -29695.682,E2 -29695.682} C_VEL
LIN {X 0,Y 155.574,Z 478.473,A -85,B 0,C 180,E1 -29698.372,E2 -29698.372} C_VEL
LIN {X 0,Y 157.571,Z 473.148,A -85,B 0,C 180,E1 -29698.917,E2 -29698.917} C_VEL
LIN {X 0,Y 158.275,Z 471.294,A -85,B 0,C 180,E1 -29698.996,E2 -29698.996} C_VEL
LIN {X 0,Y 163.848,Z 455.577,A -85,B 0,C 180,E1 -29699.431,E2 -29699.431} C_VEL
LIN {X 0,Y 168.446,Z 438.434,A -85,B 0,C 180,E1 -29699.72,E2 -29699.72} C_VEL
LIN {X 0,Y 171.527,Z 420.986,A -85,B 0,C 180,E1 -29700.022,E2 -29700.022} C_VEL
LIN {X 0,Y 174.403,Z 398.712,A -85,B 0,C 180,E1 -29700.388,E2 -29700.388} C_VEL
LIN {X 0,Y 173.201,Z 394.686,A -85,B 0,C 180,E1 -29703.742,E2 -29703.742} C_VEL
LIN {X 0,Y 172.294,Z 391.388,A -85,B 0,C 180,E1 -29707.741,E2 -29707.741} C_VEL
LIN {X 0,Y 171.842,Z 389.824,A -85,B 0,C 180,E1 -29711.8,E2 -29711.8} C_VEL
LIN {X 0,Y 171.794,Z 390.332,A -85,B 0,C 180,E1 -29714.999,E2 -29714.999} C_VEL
LIN {X 0,Y 172.392,Z 392.297,A -85,B 0,C 180,E1 -29719.588,E2 -29719.588} C_VEL
LIN {X 0,Y 173.312,Z 395.471,A -85,B 0,C 180,E1 -29723.266,E2 -29723.266} C_VEL
LIN {X 0,Y 174.322,Z 398.602,A -85,B 0,C 180,E1 -29725.96,E2 -29725.96} C_VEL
LIN {X 0,Y 170.368,Z 427.471,A -85,B 0,C 180,E1 -29726.425,E2 -29726.425} C_VEL
LIN {X 0,Y 166.471,Z 445.197,A -85,B 0,C 180,E1 -29726.789,E2 -29726.789} C_VEL
LIN {X 0,Y 161.142,Z 462.436,A -85,B 0,C 180,E1 -29727.298,E2 -29727.298} C_VEL
LIN {X 0,Y 155.091,Z 477.607,A -85,B 0,C 180,E1 -29727.914,E2 -29727.914} C_VEL
LIN {X 0,Y 147.352,Z 493.41,A -85,B 0,C 180,E1 -29728.759,E2 -29728.759} C_VEL
LIN {X 0,Y 138.67,Z 508.074,A -85,B 0,C 180,E1 -29729.781,E2 -29729.781} C_VEL
LIN {X 0,Y 129.215,Z 521.604,A -85,B 0,C 180,E1 -29731.058,E2 -29731.058} C_VEL
LIN {X 0,Y 118.937,Z 534.169,A -85,B 0,C 180,E1 -29732.644,E2 -29732.644} C_VEL
LIN {X 0,Y 107.076,Z 546.569,A -85,B 0,C 180,E1 -29734.87,E2 -29734.87} C_VEL
LIN {X 0,Y 95.363,Z 557.103,A -85,B 0,C 180,E1 -29737.603,E2 -29737.603} C_VEL
LIN {X 0,Y 82.241,Z 567.307,A -85,B 0,C 180,E1 -29741.603,E2 -29741.603} C_VEL
LIN {X 0,Y 71.137,Z 574.889,A -85,B 0,C 180,E1 -29746.244,E2 -29746.244} C_VEL
LIN {X 0,Y 59.12,Z 582.081,A -85,B 0,C 180,E1 -29753.529,E2 -29753.529} C_VEL
LIN {X 0,Y 48.306,Z 587.955,A -85,B 0,C 180,E1 -29764.119,E2 -29764.119} C_VEL
LIN {X 0,Y 39.412,Z 592.687,A -85,B 0,C 180,E1 -29779.725,E2 -29779.725} C_VEL
LIN {X 0,Y 35.238,Z 595.24,A -85,B 0,C 180,E1 -29794.282,E2 -29794.282} C_VEL
LIN {X 0,Y 33.52,Z 598.322,A -85,B 0,C 180,E1 -29823,E2 -29823} C_VEL
LIN {X 0,Y 37.42,Z 599.779,A -85,B 0,C 180,E1 -29845.705,E2 -29845.705} C_VEL
LIN {X 0,Y 44.615,Z 600.356,A -85,B 0,C 180,E1 -29861.636,E2 -29861.636} C_VEL
LIN {X 0,Y 56.441,Z 599.884,A -85,B 0,C 180,E1 -29874.942,E2 -29874.942} C_VEL
LIN {X 0,Y 70.423,Z 598.213,A -85,B 0,C 180,E1 -29883.694,E2 -29883.694} C_VEL
LIN {X 0,Y 85.506,Z 595.292,A -85,B 0,C 180,E1 -29889.501,E2 -29889.501} C_VEL
LIN {X 0,Y 93.293,Z 593.334,A -85,B 0,C 180,E1 -29891.682,E2 -29891.682} C_VEL
LIN {X 0,Y 93.436,Z 593.31,A -85,B 0,C 180,E1 -29892.098,E2 -29892.098} C_VEL
LIN {X 0,Y 80.354,Z 596.687,A -85,B 0,C 180,E1 -29895.833,E2 -29895.833} C_VEL
LIN {X 0,Y 67.773,Z 599.225,A -85,B 0,C 180,E1 -29901.053,E2 -29901.053} C_VEL
LIN {X 0,Y 50.512,Z 601.373,A -85,B 0,C 180,E1 -29913.817,E2 -29913.817} C_VEL
LIN {X 0,Y 37.9,Z 601.512,A -85,B 0,C 180,E1 -29936.204,E2 -29936.204} C_VEL
LIN {X 0,Y 34.24,Z 600.492,A -85,B 0,C 180,E1 -29958.159,E2 -29958.159} C_VEL
LIN {X 0,Y 34.155,Z 599.644,A -85,B 0,C 180,E1 -29970.003,E2 -29970.003} C_VEL
LIN {X 0,Y 34.223,Z 598.505,A -85,B 0,C 180,E1 -29981.854,E2 -29981.854} C_VEL
LIN {X 0,Y 37.888,Z 595.3,A -85,B 0,C 180,E1 -30003.817,E2 -30003.817} C_VEL
LIN {X 0,Y 45.629,Z 591.023,A -85,B 0,C 180,E1 -30020.368,E2 -30020.368} C_VEL
LIN {X 0,Y 55.781,Z 585.525,A -85,B 0,C 180,E1 -30031.881,E2 -30031.881} C_VEL
LIN {X 0,Y 67.422,Z 578.683,A -85,B 0,C 180,E1 -30039.746,E2 -30039.746} C_VEL
LIN {X 0,Y 79.938,Z 570.429,A -85,B 0,C 180,E1 -30045.265,E2 -30045.265} C_VEL
LIN {X 0,Y 91.342,Z 561.904,A -85,B 0,C 180,E1 -30048.817,E2 -30048.817} C_VEL
LIN {X 0,Y 102.991,Z 551.791,A -85,B 0,C 180,E1 -30051.677,E2 -30051.677} C_VEL
LIN {X 0,Y 114.859,Z 539.975,A -85,B 0,C 180,E1 -30053.884,E2 -30053.884} C_VEL
LIN {X 0,Y 126.011,Z 527.069,A -85,B 0,C 180,E1 -30055.518,E2 -30055.518} C_VEL
LIN {X 0,Y 136.161,Z 513.223,A -85,B 0,C 180,E1 -30056.84,E2 -30056.84} C_VEL
LIN {X 0,Y 145.137,Z 498.834,A -85,B 0,C 180,E1 -30057.766,E2 -30057.766} C_VEL
LIN {X 0,Y 152.91,Z 483.768,A -85,B 0,C 180,E1 -30058.522,E2 -30058.522} C_VEL
LIN {X 0,Y 158.275,Z 471.294,A -85,B 0,C 180,E1 -30058.996,E2 -30058.996} C_VEL
LIN {X 0,Y 159.568,Z 467.622,A -85,B 0,C 180,E1 -30059.336,E2 -30059.336} C_VEL
LIN {X 0,Y 161.011,Z 461.884,A -85,B 0,C 180,E1 -30060.533,E2 -30060.533} C_VEL
LIN {X 0,Y 162.411,Z 456.087,A -85,B 0,C 180,E1 -30061.661,E2 -30061.661} C_VEL
LIN {X 0,Y 163.411,Z 452.328,A -85,B 0,C 180,E1 -30061.925,E2 -30061.925} C_VEL
LIN {X 0,Y 167.633,Z 435.89,A -85,B 0,C 180,E1 -30062.118,E2 -30062.118} C_VEL
LIN {X 0,Y 170.577,Z 418.482,A -85,B 0,C 180,E1 -30062.402,E2 -30062.402} C_VEL
LIN {X 0,Y 172.531,Z 403.315,A -85,B 0,C 180,E1 -30062.657,E2 -30062.657} C_VEL
LIN {X 0,Y 171.657,Z 400.086,A -85,B 0,C 180,E1 -30065.832,E2 -30065.832} C_VEL
LIN {X 0,Y 171.244,Z 398.334,A -85,B 0,C 180,E1 -30068.147,E2 -30068.147} C_VEL
LIN {X 0,Y 170.88,Z 396.898,A -85,B 0,C 180,E1 -30071.867,E2 -30071.867} C_VEL
LIN {X 0,Y 170.827,Z 397.386,A -85,B 0,C 180,E1 -30074.82,E2 -30074.82} C_VEL
LIN {X 0,Y 171.324,Z 399.229,A -85,B 0,C 180,E1 -30079.158,E2 -30079.158} C_VEL
LIN {X 0,Y 172.085,Z 402.149,A -85,B 0,C 180,E1 -30082.567,E2 -30082.567} C_VEL
LIN {X 0,Y 172.452,Z 403.39,A -85,B 0,C 180,E1 -30083.738,E2 -30083.738} C_VEL
LIN {X 0,Y 168.855,Z 428.593,A -85,B 0,C 180,E1 -30084.085,E2 -30084.085} C_VEL
LIN {X 0,Y 164.959,Z 445.911,A -85,B 0,C 180,E1 -30084.395,E2 -30084.395} C_VEL
LIN {X 0,Y 159.71,Z 462.665,A -85,B 0,C 180,E1 -30084.824,E2 -30084.824} C_VEL
LIN {X 0,Y 153.132,Z 478.861,A -85,B 0,C 180,E1 -30085.37,E2 -30085.37} C_VEL
LIN {X 0,Y 146.083,Z 493.038,A -85,B 0,C 180,E1 -30086.036,E2 -30086.036} C_VEL
LIN {X 0,Y 136.95,Z 508.307,A -85,B 0,C 180,E1 -30086.919,E2 -30086.919} C_VEL
LIN {X 0,Y 127.355,Z 521.832,A -85,B 0,C 180,E1 -30087.999,E2 -30087.999} C_VEL
LIN {X 0,Y 116.91,Z 534.393,A -85,B 0,C 180,E1 -30089.347,E2 -30089.347} C_VEL
LIN {X 0,Y 106.522,Z 545.113,A -85,B 0,C 180,E1 -30090.94,E2 -30090.94} C_VEL
LIN {X 0,Y 94.491,Z 555.925,A -85,B 0,C 180,E1 -30093.201,E2 -30093.201} C_VEL
LIN {X 0,Y 82.771,Z 565.085,A -85,B 0,C 180,E1 -30096.042,E2 -30096.042} C_VEL
LIN {X 0,Y 69.289,Z 574.083,A -85,B 0,C 180,E1 -30100.47,E2 -30100.47} C_VEL
LIN {X 0,Y 56.457,Z 581.451,A -85,B 0,C 180,E1 -30106.788,E2 -30106.788} C_VEL
LIN {X 0,Y 44.532,Z 587.508,A -85,B 0,C 180,E1 -30116.468,E2 -30116.468} C_VEL
LIN {X 0,Y 36.579,Z 591.235,A -85,B 0,C 180,E1 -30127.399,E2 -30127.399} C_VEL
LIN {X 0,Y 28.132,Z 595.492,A -85,B 0,C 180,E1 -30152.148,E2 -30152.148} C_VEL
LIN {X 0,Y 26.325,Z 598.14,A -85,B 0,C 180,E1 -30182.267,E2 -30182.267} C_VEL
LIN {X 0,Y 31.629,Z 599.912,A -85,B 0,C 180,E1 -30212.714,E2 -30212.714} C_VEL
LIN {X 0,Y 42.556,Z 600.563,A -85,B 0,C 180,E1 -30232.228,E2 -30232.228} C_VEL
LIN {X 0,Y 56.332,Z 599.995,A -85,B 0,C 180,E1 -30243.598,E2 -30243.598} C_VEL
LIN {X 0,Y 73.068,Z 597.9,A -85,B 0,C 180,E1 -30251.091,E2 -30251.091} C_VEL
LIN {X 0,Y 72.069,Z 598.121,A -85,B 0,C 180,E1 -30252.805,E2 -30252.805} C_VEL
LIN {X 0,Y 59.159,Z 600.09,A -85,B 0,C 180,E1 -30258.132,E2 -30258.132} C_VEL
LIN {X 0,Y 46.04,Z 601.236,A -85,B 0,C 180,E1 -30267.255,E2 -30267.255} C_VEL
LIN {X 0,Y 36.481,Z 601.408,A -85,B 0,C 180,E1 -30279.599,E2 -30279.599} C_VEL
LIN {X 0,Y 29.042,Z 600.812,A -85,B 0,C 180,E1 -30301.059,E2 -30301.059} C_VEL
LIN {X 0,Y 27.035,Z 599.209,A -85,B 0,C 180,E1 -30330.004,E2 -30330.004} C_VEL
LIN {X 0,Y 29.026,Z 596.536,A -85,B 0,C 180,E1 -30358.968,E2 -30358.968} C_VEL
LIN {X 0,Y 36.441,Z 592.662,A -85,B 0,C 180,E1 -30380.487,E2 -30380.487} C_VEL
LIN {X 0,Y 46.885,Z 587.669,A -85,B 0,C 180,E1 -30394.083,E2 -30394.083} C_VEL
LIN {X 0,Y 58.903,Z 581.402,A -85,B 0,C 180,E1 -30402.656,E2 -30402.656} C_VEL
LIN {X 0,Y 71.775,Z 573.713,A -85,B 0,C 180,E1 -30408.289,E2 -30408.289} C_VEL
LIN {X 0,Y 85.138,Z 564.505,A -85,B 0,C 180,E1 -30412.136,E2 -30412.136} C_VEL
LIN {X 0,Y 97.038,Z 554.957,A -85,B 0,C 180,E1 -30414.782,E2 -30414.782} C_VEL
LIN {X 0,Y 109.106,Z 543.747,A -85,B 0,C 180,E1 -30416.786,E2 -30416.786} C_VEL
LIN {X 0,Y 119.538,Z 532.479,A -85,B 0,C 180,E1 -30418.154,E2 -30418.154} C_VEL
LIN {X 0,Y 130.028,Z 519.377,A -85,B 0,C 180,E1 -30419.296,E2 -30419.296} C_VEL
LIN {X 0,Y 138.452,Z 507.189,A -85,B 0,C 180,E1 -30420.076,E2 -30420.076} C_VEL
LIN {X 0,Y 146.723,Z 492.975,A -85,B 0,C 180,E1 -30420.768,E2 -30420.768} C_VEL
LIN {X 0,Y 154.219,Z 477.482,A -85,B 0,C 180,E1 -30421.338,E2 -30421.338} C_VEL
LIN {X 0,Y 160.403,Z 461.645,A -85,B 0,C 180,E1 -30421.772,E2 -30421.772} C_VEL
LIN {X 0,Y 163.411,Z 452.328,A -85,B 0,C 180,E1 -30421.925,E2 -30421.925} C_VEL
LIN {X 0,Y 164.984,Z 446.672,A -85,B 0,C 180,E1 -30422.142,E2 -30422.142} C_VEL
LIN {X 0,Y 166.765,Z 437.438,A -85,B 0,C 180,E1 -30423.238,E2 -30423.238} C_VEL
LIN {X 0,Y 168.166,Z 428.118,A -85,B 0,C 180,E1 -30424.382,E2 -30424.382} C_VEL
LIN {X 0,Y 168.964,Z 422.306,A -85,B 0,C 180,E1 -30424.712,E2 -30424.712} C_VEL
LIN {X 0,Y 170.866,Z 408.302,A -85,B 0,C 180,E1 -30424.897,E2 -30424.897} C_VEL
LIN {X 0,Y 170.214,Z 405.291,A -85,B 0,C 180,E1 -30428.504,E2 -30428.504} C_VEL
LIN {X 0,Y 169.918,Z 403.972,A -85,B 0,C 180,E1 -30431.935,E2 -30431.935} C_VEL
LIN {X 0,Y 169.866,Z 404.38,A -85,B 0,C 180,E1 -30434.576,E2 -30434.576} C_VEL
LIN {X 0,Y 170.277,Z 406.178,A -85,B 0,C 180,E1 -30438.786,E2 -30438.786} C_VEL
LIN {X 0,Y 170.788,Z 408.393,A -85,B 0,C 180,E1 -30441.444,E2 -30441.444} C_VEL
LIN {X 0,Y 167.74,Z 429.043,A -85,B 0,C 180,E1 -30441.703,E2 -30441.703} C_VEL
LIN {X 0,Y 163.821,Z 446.237,A -85,B 0,C 180,E1 -30441.956,E2 -30441.956} C_VEL
LIN {X 0,Y 158.575,Z 462.823,A -85,B 0,C 180,E1 -30442.306,E2 -30442.306} C_VEL
LIN {X 0,Y 152.395,Z 478.002,A -85,B 0,C 180,E1 -30442.729,E2 -30442.729} C_VEL
LIN {X 0,Y 144.698,Z 493.423,A -85,B 0,C 180,E1 -30443.3,E2 -30443.3} C_VEL
LIN {X 0,Y 135.587,Z 508.482,A -85,B 0,C 180,E1 -30443.996,E2 -30443.996} C_VEL
LIN {X 0,Y 125.871,Z 522.014,A -85,B 0,C 180,E1 -30444.862,E2 -30444.862} C_VEL
LIN {X 0,Y 115.33,Z 534.519,A -85,B 0,C 180,E1 -30445.936,E2 -30445.936} C_VEL
LIN {X 0,Y 104.715,Z 545.303,A -85,B 0,C 180,E1 -30447.216,E2 -30447.216} C_VEL
LIN {X 0,Y 92.447,Z 556.114,A -85,B 0,C 180,E1 -30449.042,E2 -30449.042} C_VEL
LIN {X 0,Y 80.441,Z 565.265,A -85,B 0,C 180,E1 -30451.344,E2 -30451.344} C_VEL
LIN {X 0,Y 66.468,Z 574.28,A -85,B 0,C 180,E1 -30454.969,E2 -30454.969} C_VEL
LIN {X 0,Y 54.668,Z 580.801,A -85,B 0,C 180,E1 -30459.523,E2 -30459.523} C_VEL
LIN {X 0,Y 41.685,Z 587.053,A -85,B 0,C 180,E1 -30467.59,E2 -30467.59} C_VEL
LIN {X 0,Y 29.788,Z 592.013,A -85,B 0,C 180,E1 -30481.84,E2 -30481.84} C_VEL
LIN {X 0,Y 20.837,Z 595.866,A -85,B 0,C 180,E1 -30509.994,E2 -30509.994} C_VEL
LIN {X 0,Y 20.024,Z 598.667,A -85,B 0,C 180,E1 -30554.576,E2 -30554.576} C_VEL
LIN {X 0,Y 28.782,Z 600.286,A -85,B 0,C 180,E1 -30587.591,E2 -30587.591} C_VEL
LIN {X 0,Y 42.252,Z 600.762,A -85,B 0,C 180,E1 -30603.663,E2 -30603.663} C_VEL
LIN {X 0,Y 55.75,Z 600.208,A -85,B 0,C 180,E1 -30611.403,E2 -30611.403} C_VEL
LIN {X 0,Y 50.754,Z 600.632,A -85,B 0,C 180,E1 -30614.247,E2 -30614.247} C_VEL
LIN {X 0,Y 38.167,Z 601.237,A -85,B 0,C 180,E1 -30622.982,E2 -30622.982} C_VEL
LIN {X 0,Y 27.176,Z 600.893,A -85,B 0,C 180,E1 -30639.127,E2 -30639.127} C_VEL
LIN {X 0,Y 20.484,Z 599.747,A -85,B 0,C 180,E1 -30669.94,E2 -30669.94} C_VEL
LIN {X 0,Y 19.931,Z 598.771,A -85,B 0,C 180,E1 -30690.006,E2 -30690.006} C_VEL
LIN {X 0,Y 23.023,Z 595.962,A -85,B 0,C 180,E1 -30727.633,E2 -30727.633} C_VEL
LIN {X 0,Y 32.339,Z 592.006,A -85,B 0,C 180,E1 -30750.383,E2 -30750.383} C_VEL
LIN {X 0,Y 44.209,Z 586.86,A -85,B 0,C 180,E1 -30762.528,E2 -30762.528} C_VEL
LIN {X 0,Y 57.163,Z 580.488,A -85,B 0,C 180,E1 -30769.606,E2 -30769.606} C_VEL
LIN {X 0,Y 72.065,Z 571.798,A -85,B 0,C 180,E1 -30774.404,E2 -30774.404} C_VEL
LIN {X 0,Y 86.186,Z 561.978,A -85,B 0,C 180,E1 -30777.353,E2 -30777.353} C_VEL
LIN {X 0,Y 99.691,Z 550.832,A -85,B 0,C 180,E1 -30779.492,E2 -30779.492} C_VEL
LIN {X 0,Y 110.702,Z 540.249,A -85,B 0,C 180,E1 -30780.786,E2 -30780.786} C_VEL
LIN {X 0,Y 122.174,Z 527.48,A -85,B 0,C 180,E1 -30781.826,E2 -30781.826} C_VEL
LIN {X 0,Y 131.915,Z 514.778,A -85,B 0,C 180,E1 -30782.635,E2 -30782.635} C_VEL
LIN {X 0,Y 141.668,Z 499.67,A -85,B 0,C 180,E1 -30783.262,E2 -30783.262} C_VEL
LIN {X 0,Y 149.665,Z 484.688,A -85,B 0,C 180,E1 -30783.75,E2 -30783.75} C_VEL
LIN {X 0,Y 156.336,Z 469.481,A -85,B 0,C 180,E1 -30784.111,E2 -30784.111} C_VEL
LIN {X 0,Y 161.896,Z 453.617,A -85,B 0,C 180,E1 -30784.375,E2 -30784.375} C_VEL
LIN {X 0,Y 166.317,Z 436.976,A -85,B 0,C 180,E1 -30784.513,E2 -30784.513} C_VEL
LIN {X 0,Y 168.964,Z 422.306,A -85,B 0,C 180,E1 -30784.712,E2 -30784.712} C_VEL
LIN {X 0,Y 169.268,Z 419.836,A -85,B 0,C 180,E1 -30784.95,E2 -30784.95} C_VEL
LIN {X 0,Y 169.41,Z 416.751,A -85,B 0,C 180,E1 -30785.8,E2 -30785.8} C_VEL
LIN {X 0,Y 169.357,Z 414.522,A -85,B 0,C 180,E1 -30786.963,E2 -30786.963} C_VEL
LIN {X 0,Y 169.15,Z 412.498,A -85,B 0,C 180,E1 -30788.9,E2 -30788.9} C_VEL
LIN {X 0,Y 168.975,Z 411.48,A -85,B 0,C 180,E1 -30790.935,E2 -30790.935} C_VEL
LIN {X 0,Y 168.957,Z 411.036,A -85,B 0,C 180,E1 -30792.004,E2 -30792.004} C_VEL
LIN {X 0,Y 168.904,Z 411.443,A -85,B 0,C 180,E1 -30794.457,E2 -30794.457} C_VEL
LIN {X 0,Y 169.201,Z 412.933,A -85,B 0,C 180,E1 -30798.152,E2 -30798.152} C_VEL
LIN {X 0,Y 169.339,Z 413.719,A -85,B 0,C 180,E1 -30799.109,E2 -30799.109} C_VEL
LIN {X 0,Y 167.141,Z 428.307,A -85,B 0,C 180,E1 -30799.284,E2 -30799.284} C_VEL
LIN {X 0,Y 163.135,Z 445.989,A -85,B 0,C 180,E1 -30799.48,E2 -30799.48} C_VEL
LIN {X 0,Y 157.696,Z 463.099,A -85,B 0,C 180,E1 -30799.755,E2 -30799.755} C_VEL
LIN {X 0,Y 151.072,Z 479.156,A -85,B 0,C 180,E1 -30800.092,E2 -30800.092} C_VEL
LIN {X 0,Y 143.519,Z 494.023,A -85,B 0,C 180,E1 -30800.523,E2 -30800.523} C_VEL
LIN {X 0,Y 134.584,Z 508.642,A -85,B 0,C 180,E1 -30801.022,E2 -30801.022} C_VEL
LIN {X 0,Y 124.778,Z 522.179,A -85,B 0,C 180,E1 -30801.666,E2 -30801.666} C_VEL
LIN {X 0,Y 114.065,Z 534.752,A -85,B 0,C 180,E1 -30802.449,E2 -30802.449} C_VEL
LIN {X 0,Y 101.6,Z 547.155,A -85,B 0,C 180,E1 -30803.573,E2 -30803.573} C_VEL
LIN {X 0,Y 89.145,Z 557.692,A -85,B 0,C 180,E1 -30804.955,E2 -30804.955} C_VEL
LIN {X 0,Y 74.934,Z 567.9,A -85,B 0,C 180,E1 -30807,E2 -30807} C_VEL
LIN {X 0,Y 60.804,Z 576.432,A -85,B 0,C 180,E1 -30809.9,E2 -30809.9} C_VEL
LIN {X 0,Y 46.832,Z 583.518,A -85,B 0,C 180,E1 -30814.369,E2 -30814.369} C_VEL
LIN {X 0,Y 33.198,Z 589.215,A -85,B 0,C 180,E1 -30822.183,E2 -30822.183} C_VEL
LIN {X 0,Y 23.402,Z 592.781,A -85,B 0,C 180,E1 -30833.079,E2 -30833.079} C_VEL
LIN {X 0,Y 13.091,Z 596.467,A -85,B 0,C 180,E1 -30869.991,E2 -30869.991} C_VEL
LIN {X 0,Y 14.344,Z 598.905,A -85,B 0,C 180,E1 -30930.663,E2 -30930.663} C_VEL
LIN {X 0,Y 24.624,Z 600.353,A -85,B 0,C 180,E1 -30960,E2 -30960} C_VEL
LIN {X 0,Y 36.499,Z 600.981,A -85,B 0,C 180,E1 -30971.102,E2 -30971.102} C_VEL
LIN {X 0,Y 35.974,Z 600.994,A -85,B 0,C 180,E1 -30972.378,E2 -30972.378} C_VEL
LIN {X 0,Y 23.326,Z 600.579,A -85,B 0,C 180,E1 -30985.341,E2 -30985.341} C_VEL
LIN {X 0,Y 13.983,Z 599.342,A -85,B 0,C 180,E1 -31019.837,E2 -31019.837} C_VEL
LIN {X 0,Y 12.812,Z 598.326,A -85,B 0,C 180,E1 -31050.009,E2 -31050.009} C_VEL
LIN {X 0,Y 17.899,Z 595.378,A -85,B 0,C 180,E1 -31101.756,E2 -31101.756} C_VEL
LIN {X 0,Y 29.447,Z 591.347,A -85,B 0,C 180,E1 -31122.692,E2 -31122.692} C_VEL
LIN {X 0,Y 42.597,Z 586.048,A -85,B 0,C 180,E1 -31131.871,E2 -31131.871} C_VEL
LIN {X 0,Y 56.309,Z 579.515,A -85,B 0,C 180,E1 -31136.866,E2 -31136.866} C_VEL
LIN {X 0,Y 70.646,Z 571.357,A -85,B 0,C 180,E1 -31140,E2 -31140} C_VEL
LIN {X 0,Y 84.386,Z 561.996,A -85,B 0,C 180,E1 -31141.956,E2 -31141.956} C_VEL
LIN {X 0,Y 96.803,Z 552.021,A -85,B 0,C 180,E1 -31143.37,E2 -31143.37} C_VEL
LIN {X 0,Y 109.257,Z 540.362,A -85,B 0,C 180,E1 -31144.404,E2 -31144.404} C_VEL
LIN {X 0,Y 120.835,Z 527.655,A -85,B 0,C 180,E1 -31145.109,E2 -31145.109} C_VEL
LIN {X 0,Y 131.553,Z 513.733,A -85,B 0,C 180,E1 -31145.727,E2 -31145.727} C_VEL
LIN {X 0,Y 140.574,Z 499.811,A -85,B 0,C 180,E1 -31146.105,E2 -31146.105} C_VEL
LIN {X 0,Y 148.526,Z 485.095,A -85,B 0,C 180,E1 -31146.443,E2 -31146.443} C_VEL
LIN {X 0,Y 155.68,Z 468.922,A -85,B 0,C 180,E1 -31146.703,E2 -31146.703} C_VEL
LIN {X 0,Y 161.266,Z 452.942,A -85,B 0,C 180,E1 -31146.875,E2 -31146.875} C_VEL
LIN {X 0,Y 165.634,Z 436.414,A -85,B 0,C 180,E1 -31146.941,E2 -31146.941} C_VEL
LIN {X 0,Y 168.742,Z 418.686,A -85,B 0,C 180,E1 -31147.152,E2 -31147.152} C_VEL
LIN {X 0,Y 169.424,Z 413.468,A -85,B 0,C 180,E1 -31147.258,E2 -31147.258} C_VEL
LIN {X 0,Y 169.135,Z 412.135,A -85,B 0,C 180,E1 -31149.218,E2 -31149.218} C_VEL
LIN {X 0,Y 168.975,Z 411.48,A -85,B 0,C 180,E1 -31150.935,E2 -31150.935} C_VEL
LIN {X 0,Y 168.842,Z 412.011,A -85,B 0,C 180,E1 -31151.719,E2 -31151.719} C_VEL
LIN {X 0,Y 168.444,Z 414.681,A -85,B 0,C 180,E1 -31152.805,E2 -31152.805} C_VEL
LIN {X 0,Y 168.048,Z 417.668,A -85,B 0,C 180,E1 -31153.886,E2 -31153.886} C_VEL
LIN {X 0,Y 167.941,Z 418.621,A -85,B 0,C 180,E1 -31154.682,E2 -31154.682} C_VEL
LIN {X 0,Y 168.043,Z 419.37,A -85,B 0,C 180,E1 -31156.773,E2 -31156.773} C_VEL
LIN {X 0,Y 164.883,Z 436.813,A -85,B 0,C 180,E1 -31156.924,E2 -31156.924} C_VEL
LIN {X 0,Y 160.356,Z 453.579,A -85,B 0,C 180,E1 -31157.063,E2 -31157.063} C_VEL
LIN {X 0,Y 154.985,Z 468.663,A -85,B 0,C 180,E1 -31157.233,E2 -31157.233} C_VEL
LIN {X 0,Y 148.292,Z 483.803,A -85,B 0,C 180,E1 -31157.487,E2 -31157.487} C_VEL
LIN {X 0,Y 140.239,Z 498.758,A -85,B 0,C 180,E1 -31157.791,E2 -31157.791} C_VEL
LIN {X 0,Y 131.249,Z 512.645,A -85,B 0,C 180,E1 -31158.11,E2 -31158.11} C_VEL
LIN {X 0,Y 121.381,Z 525.535,A -85,B 0,C 180,E1 -31158.536,E2 -31158.536} C_VEL
LIN {X 0,Y 110.31,Z 537.913,A -85,B 0,C 180,E1 -31159.04,E2 -31159.04} C_VEL
LIN {X 0,Y 98.901,Z 548.899,A -85,B 0,C 180,E1 -31159.684,E2 -31159.684} C_VEL
LIN {X 0,Y 86.305,Z 559.217,A -85,B 0,C 180,E1 -31160.531,E2 -31160.531} C_VEL
LIN {X 0,Y 73.713,Z 568.028,A -85,B 0,C 180,E1 -31161.626,E2 -31161.626} C_VEL
LIN {X 0,Y 61.095,Z 575.632,A -85,B 0,C 180,E1 -31163.032,E2 -31163.032} C_VEL
LIN {X 0,Y 46.696,Z 582.834,A -85,B 0,C 180,E1 -31165.437,E2 -31165.437} C_VEL
LIN {X 0,Y 32.326,Z 588.723,A -85,B 0,C 180,E1 -31169.577,E2 -31169.577} C_VEL
LIN {X 0,Y 17.93,Z 593.479,A -85,B 0,C 180,E1 -31178.366,E2 -31178.366} C_VEL
LIN {X 0,Y 8.02,Z 596.176,A -85,B 0,C 180,E1 -31201.201,E2 -31201.201} C_VEL
LIN {X 0,Y 10.526,Z 599.084,A -85,B 0,C 180,E1 -31320,E2 -31320} C_VEL
LIN {X 0,Y 14.194,Z 599.566,A -85,B 0,C 180,E1 -31328.074,E2 -31328.074} C_VEL
LIN {X 0,Y 14.599,Z 599.671,A -85,B 0,C 180,E1 -31335.711,E2 -31335.711} C_VEL
LIN {X 0,Y 5.686,Z 597.871,A -85,B 0,C 180,E1 -31410.021,E2 -31410.021} C_VEL
LIN {X 0,Y 14.593,Z 594.771,A -85,B 0,C 180,E1 -31484.439,E2 -31484.439} C_VEL
LIN {X 0,Y 28.156,Z 590.621,A -85,B 0,C 180,E1 -31496.855,E2 -31496.855} C_VEL
LIN {X 0,Y 42.186,Z 585.2,A -85,B 0,C 180,E1 -31501.617,E2 -31501.617} C_VEL
LIN {X 0,Y 56.379,Z 578.492,A -85,B 0,C 180,E1 -31504.227,E2 -31504.227} C_VEL
LIN {X 0,Y 70.645,Z 570.384,A -85,B 0,C 180,E1 -31505.821,E2 -31505.821} C_VEL
LIN {X 0,Y 84.944,Z 560.659,A -85,B 0,C 180,E1 -31506.855,E2 -31506.855} C_VEL
LIN {X 0,Y 97.498,Z 550.475,A -85,B 0,C 180,E1 -31507.628,E2 -31507.628} C_VEL
LIN {X 0,Y 110.052,Z 538.55,A -85,B 0,C 180,E1 -31508.171,E2 -31508.171} C_VEL
LIN {X 0,Y 121.7,Z 525.518,A -85,B 0,C 180,E1 -31508.528,E2 -31508.528} C_VEL
LIN {X 0,Y 131.574,Z 512.531,A -85,B 0,C 180,E1 -31508.821,E2 -31508.821} C_VEL
LIN {X 0,Y 140.534,Z 498.66,A -85,B 0,C 180,E1 -31509.005,E2 -31509.005} C_VEL
LIN {X 0,Y 148.62,Z 483.523,A -85,B 0,C 180,E1 -31509.196,E2 -31509.196} C_VEL
LIN {X 0,Y 155.341,Z 468.144,A -85,B 0,C 180,E1 -31509.302,E2 -31509.302} C_VEL
LIN {X 0,Y 160.947,Z 451.953,A -85,B 0,C 180,E1 -31509.393,E2 -31509.393} C_VEL
LIN {X 0,Y 165.277,Z 435.262,A -85,B 0,C 180,E1 -31509.408,E2 -31509.408} C_VEL
LIN {X 0,Y 168.021,Z 419.813,A -85,B 0,C 180,E1 -31509.548,E2 -31509.548} C_VEL
LIN {X 0,Y 168.123,Z 419.056,A -85,B 0,C 180,E1 -31509.626,E2 -31509.626} C_VEL
LIN {X 0,Y 167.996,Z 418.106,A -85,B 0,C 180,E1 -31512.074,E2 -31512.074} C_VEL
LIN {X 0,Y 167.942,Z 418.568,A -85,B 0,C 180,E1 -31514.542,E2 -31514.542} C_VEL
LIN {X 0,Y 167.941,Z 418.621,A -85,B 0,C 180,E1 -31514.682,E2 -31514.682} C_VEL
LIN {X 0,Y 167.827,Z 419.601,A -85,B 0,C 180,E1 -31515.161,E2 -31515.161} C_VEL
LIN {X 0,Y 167.509,Z 421.848,A -85,B 0,C 180,E1 -31515.439,E2 -31515.439} C_VEL
LIN {X 0,Y 166.906,Z 425.608,A -85,B 0,C 180,E1 -31515.393,E2 -31515.393} C_VEL
LIN {X 0,Y 164.75,Z 436.34,A -85,B 0,C 180,E1 -31514.53,E2 -31514.53} C_VEL
LIN {X 0,Y 163.983,Z 439.54,A -85,B 0,C 180,E1 -31514.465,E2 -31514.465} C_VEL
LIN {X 0,Y 159.296,Z 456.213,A -85,B 0,C 180,E1 -31514.565,E2 -31514.565} C_VEL
LIN {X 0,Y 153.002,Z 473.061,A -85,B 0,C 180,E1 -31514.651,E2 -31514.651} C_VEL
LIN {X 0,Y 145.39,Z 489.121,A -85,B 0,C 180,E1 -31514.81,E2 -31514.81} C_VEL
LIN {X 0,Y 137.358,Z 503.037,A -85,B 0,C 180,E1 -31514.925,E2 -31514.925} C_VEL
LIN {X 0,Y 127.375,Z 517.589,A -85,B 0,C 180,E1 -31515.078,E2 -31515.078} C_VEL
